(* Logix 5000 project; controller VET 1756-L62 rev 19.52; software revision 19.01; part 9 of 27 *)

        [46].Data.peso_f[8] := 50.0, [46].Data.peso_f[9] := 43.6, [46].Data.peso_f[10] := 35.0, [46].Data.peso_f[11] := 12.0, [46].Data.peso_f[12] := 60.0, [46].Data.peso_f[13] := 56.0, [46].Data.peso_f[14] := 25.0, [46].Data.peso_f[15] := 90.0, [46].Data.peso_r[0] := 332.00415, [46].Data.peso_r[1] := 319.90973, [46].Data.peso_r[2] := 285.3365, [46].Data.peso_r[3] := 180.5769, [46].Data.peso_r[4] := 159.76408, [46].Data.peso_r[5] := 109.9774, [46].Data.peso_r[6] := 90.60315, [46].Data.peso_r[7] := 90.27219, [46].Data.peso_r[8] := 50.001286, [46].Data.peso_r[9] := 43.602726, [46].Data.peso_r[10] := 34.989906, [46].Data.peso_r[11] := 11.96817, [46].Data.peso_r[12] := 59.986206, [46].Data.peso_r[13] := 56.00316, [46].Data.peso_r[14] := 25.010452, [46].Data.peso_r[15] := 89.91622, [46].Data.tolva[0] := 3, [46].Data.tolva[1] := 4, [46].Data.tolva[2] := 10, [46].Data.tolva[3] := 12, [46].Data.tolva[4] := 6, [46].Data.tolva[5] := 7, [46].Data.tolva[6] := 14, [46].Data.tolva[7] := 15, [46].Data.tolva[8] := 18, [46].Data.tolva[9] := 20, [46].Data.tolva[10] := 22, [46].Data.tolva[11] := 24, [46].Data.tolva[12] := 27, [46].Data.tolva[13] := 29, [46].Data.tolva[14] := 31, [46].Data.tolva[15] := 38, [46].Data.lugar[0] := 1, [46].Data.lugar[1] := 1, [46].Data.lugar[2] := 1, [46].Data.lugar[3] := 1, [46].Data.lugar[4] := 2, [46].Data.lugar[5] := 2, [46].Data.lugar[6] := 2, [46].Data.lugar[7] := 2, [46].Data.lugar[8] := 3, [46].Data.lugar[9] := 3, [46].Data.lugar[10] := 3, [46].Data.lugar[11] := 3, [46].Data.lugar[12] := 4, [46].Data.lugar[13] := 4, [46].Data.lugar[14] := 4, [46].Data.lugar[15] := 6, [46].Data.flags[0] := 5, [46].Data.flags[1] := 5, [46].Data.flags[2] := 5, [46].Data.flags[3] := 5,
        [46].Data.flags[4] := 5, [46].Data.flags[5] := 5, [46].Data.flags[6] := 5, [46].Data.flags[7] := 5, [46].Data.flags[8] := 5, [46].Data.flags[9] := 5, [46].Data.flags[10] := 5, [46].Data.flags[11] := 5, [46].Data.flags[12] := 5, [46].Data.flags[13] := 5, [46].Data.flags[14] := 5, [46].Data.flags[15] := 5, [46].Data.fecha_i[0] := 19980102, [46].Data.fecha_i[1] := 19980102, [46].Data.fecha_i[2] := 19980102, [46].Data.fecha_i[3] := 19980102, [46].Data.fecha_i[4] := 19980102, [46].Data.fecha_i[5] := 19980102, [46].Data.fecha_i[6] := 19980102, [46].Data.fecha_i[7] := 19980102, [46].Data.fecha_i[8] := 19980102, [46].Data.fecha_i[9] := 19980102, [46].Data.fecha_i[10] := 19980102, [46].Data.fecha_i[11] := 19980102, [46].Data.fecha_i[12] := 19980102, [46].Data.fecha_i[13] := 19980102, [46].Data.fecha_i[14] := 19980102, [46].Data.fecha_i[15] := 19980102, [46].Data.fecha_f[0] := 19980102, [46].Data.fecha_f[1] := 19980102, [46].Data.fecha_f[2] := 19980102, [46].Data.fecha_f[3] := 19980102, [46].Data.fecha_f[4] := 19980102, [46].Data.fecha_f[5] := 19980102, [46].Data.fecha_f[6] := 19980102, [46].Data.fecha_f[7] := 19980102, [46].Data.fecha_f[8] := 19980102, [46].Data.fecha_f[9] := 19980102, [46].Data.fecha_f[10] := 19980102, [46].Data.fecha_f[11] := 19980102, [46].Data.fecha_f[12] := 19980102, [46].Data.fecha_f[13] := 19980102, [46].Data.fecha_f[14] := 19980102, [46].Data.fecha_f[15] := 19980102, [46].Data.hora_i[0] := 22451016, [46].Data.hora_i[1] := 22452601, [46].Data.hora_i[2] := 22454141, [46].Data.hora_i[3] := 22455546, [46].Data.hora_i[4] := 22451016, [46].Data.hora_i[5] := 22452781, [46].Data.hora_i[6] := 22453811, [46].Data.hora_i[7] := 22455416, [46].Data.hora_i[8] := 22451016, [46].Data.hora_i[9] := 22465331, [46].Data.hora_i[10] := 22482366, [46].Data.hora_i[11] := 22493681, [46].Data.hora_i[12] := 22451016, [46].Data.hora_i[13] := 22471706, [46].Data.hora_i[14] := 22491621, [46].Data.hora_i[15] := 22503341,
        [46].Data.hora_f[0] := 22452581, [46].Data.hora_f[1] := 22454121, [46].Data.hora_f[2] := 22455526, [46].Data.hora_f[3] := 22460531, [46].Data.hora_f[4] := 22452761, [46].Data.hora_f[5] := 22453791, [46].Data.hora_f[6] := 22455396, [46].Data.hora_f[7] := 22460296, [46].Data.hora_f[8] := 22465311, [46].Data.hora_f[9] := 22482346, [46].Data.hora_f[10] := 22493661, [46].Data.hora_f[11] := 22500376, [46].Data.hora_f[12] := 22471686, [46].Data.hora_f[13] := 22491601, [46].Data.hora_f[14] := 22501286, [46].Data.hora_f[15] := 22512556, [47].Head.folio := 48, [47].Head.orden := -4, [47].Head.formula := 'DUMMY$00$00$00$00$00', [47].Head.correlativo := 8, [47].Head.total_batch := 10, [47].Head.peso_teorico := 1939.6, [47].Data.codigo[0] := 51, [47].Data.codigo[1] := 53, [47].Data.codigo[2] := 55, [47].Data.codigo[3] := 57, [47].Data.codigo[4] := 59, [47].Data.codigo[5] := 60, [47].Data.codigo[6] := 63, [47].Data.codigo[7] := 64, [47].Data.codigo[8] := 67, [47].Data.codigo[9] := 69, [47].Data.codigo[10] := 71, [47].Data.codigo[11] := 73, [47].Data.codigo[12] := 75, [47].Data.codigo[13] := 77, [47].Data.codigo[14] := 79, [47].Data.codigo[15] := 81, [47].Data.peso_f[0] := 333.0, [47].Data.peso_f[1] := 320.0, [47].Data.peso_f[2] := 285.0, [47].Data.peso_f[3] := 180.0, [47].Data.peso_f[4] := 160.0, [47].Data.peso_f[5] := 110.0, [47].Data.peso_f[6] := 90.0, [47].Data.peso_f[7] := 90.0, [47].Data.peso_f[8] := 50.0, [47].Data.peso_f[9] := 43.6, [47].Data.peso_f[10] := 35.0, [47].Data.peso_f[11] := 12.0, [47].Data.peso_f[12] := 60.0, [47].Data.peso_f[13] := 56.0, [47].Data.peso_f[14] := 25.0, [47].Data.peso_f[15] := 90.0, [47].Data.peso_r[0] := 334.1721, [47].Data.peso_r[1] := 319.58975, [47].Data.peso_r[2] := 284.6056, [47].Data.peso_r[3] := 180.28247, [47].Data.peso_r[4] := 159.7642, [47].Data.peso_r[5] := 109.9774,
        [47].Data.peso_r[6] := 90.59973, [47].Data.peso_r[7] := 91.76578, [47].Data.peso_r[8] := 50.000805, [47].Data.peso_r[9] := 43.602703, [47].Data.peso_r[10] := 34.989876, [47].Data.peso_r[11] := 12.01152, [47].Data.peso_r[12] := 60.010212, [47].Data.peso_r[13] := 56.003162, [47].Data.peso_r[14] := 25.01043, [47].Data.peso_r[15] := 90.216225, [47].Data.tolva[0] := 3, [47].Data.tolva[1] := 4, [47].Data.tolva[2] := 10, [47].Data.tolva[3] := 12, [47].Data.tolva[4] := 6, [47].Data.tolva[5] := 7, [47].Data.tolva[6] := 14, [47].Data.tolva[7] := 15, [47].Data.tolva[8] := 18, [47].Data.tolva[9] := 20, [47].Data.tolva[10] := 22, [47].Data.tolva[11] := 24, [47].Data.tolva[12] := 27, [47].Data.tolva[13] := 29, [47].Data.tolva[14] := 31, [47].Data.tolva[15] := 38, [47].Data.lugar[0] := 1, [47].Data.lugar[1] := 1, [47].Data.lugar[2] := 1, [47].Data.lugar[3] := 1, [47].Data.lugar[4] := 2, [47].Data.lugar[5] := 2, [47].Data.lugar[6] := 2, [47].Data.lugar[7] := 2, [47].Data.lugar[8] := 3, [47].Data.lugar[9] := 3, [47].Data.lugar[10] := 3, [47].Data.lugar[11] := 3, [47].Data.lugar[12] := 4, [47].Data.lugar[13] := 4, [47].Data.lugar[14] := 4, [47].Data.lugar[15] := 6, [47].Data.flags[0] := 5, [47].Data.flags[1] := 5, [47].Data.flags[2] := 5, [47].Data.flags[3] := 5, [47].Data.flags[4] := 5, [47].Data.flags[5] := 5, [47].Data.flags[6] := 5, [47].Data.flags[7] := 5, [47].Data.flags[8] := 5, [47].Data.flags[9] := 5, [47].Data.flags[10] := 5, [47].Data.flags[11] := 5, [47].Data.flags[12] := 5, [47].Data.flags[13] := 5, [47].Data.flags[14] := 5, [47].Data.flags[15] := 5, [47].Data.fecha_i[0] := 19980102, [47].Data.fecha_i[1] := 19980102,
        [47].Data.fecha_i[2] := 19980102, [47].Data.fecha_i[3] := 19980102, [47].Data.fecha_i[4] := 19980102, [47].Data.fecha_i[5] := 19980102, [47].Data.fecha_i[6] := 19980102, [47].Data.fecha_i[7] := 19980102, [47].Data.fecha_i[8] := 19980102, [47].Data.fecha_i[9] := 19980102, [47].Data.fecha_i[10] := 19980102, [47].Data.fecha_i[11] := 19980102, [47].Data.fecha_i[12] := 19980102, [47].Data.fecha_i[13] := 19980102, [47].Data.fecha_i[14] := 19980102, [47].Data.fecha_i[15] := 19980102, [47].Data.fecha_f[0] := 19980102, [47].Data.fecha_f[1] := 19980102, [47].Data.fecha_f[2] := 19980102, [47].Data.fecha_f[3] := 19980102, [47].Data.fecha_f[4] := 19980102, [47].Data.fecha_f[5] := 19980102, [47].Data.fecha_f[6] := 19980102, [47].Data.fecha_f[7] := 19980102, [47].Data.fecha_f[8] := 19980102, [47].Data.fecha_f[9] := 19980102, [47].Data.fecha_f[10] := 19980102, [47].Data.fecha_f[11] := 19980102, [47].Data.fecha_f[12] := 19980102, [47].Data.fecha_f[13] := 19980102, [47].Data.fecha_f[14] := 19980102, [47].Data.fecha_f[15] := 19980102, [47].Data.hora_i[0] := 22522096, [47].Data.hora_i[1] := 22523686, [47].Data.hora_i[2] := 22525226, [47].Data.hora_i[3] := 22530631, [47].Data.hora_i[4] := 22522096, [47].Data.hora_i[5] := 22523861, [47].Data.hora_i[6] := 22524891, [47].Data.hora_i[7] := 22541271, [47].Data.hora_i[8] := 22522096, [47].Data.hora_i[9] := 22540411, [47].Data.hora_i[10] := 22553446, [47].Data.hora_i[11] := 22564761, [47].Data.hora_i[12] := 22522096, [47].Data.hora_i[13] := 22542786, [47].Data.hora_i[14] := 22562701, [47].Data.hora_i[15] := 22574421, [47].Data.hora_f[0] := 22523666, [47].Data.hora_f[1] := 22525206, [47].Data.hora_f[2] := 22530611, [47].Data.hora_f[3] := 22531616, [47].Data.hora_f[4] := 22523841, [47].Data.hora_f[5] := 22524871, [47].Data.hora_f[6] := 22541251, [47].Data.hora_f[7] := 22543396, [47].Data.hora_f[8] := 22540391, [47].Data.hora_f[9] := 22553426, [47].Data.hora_f[10] := 22564741, [47].Data.hora_f[11] := 22571461, [47].Data.hora_f[12] := 22542766, [47].Data.hora_f[13] := 22562681,
        [47].Data.hora_f[14] := 22572366, [47].Data.hora_f[15] := 22583656, [48].Head.folio := 49, [48].Head.orden := -4, [48].Head.formula := 'DUMMY$00$00$00$00$00', [48].Head.correlativo := 9, [48].Head.total_batch := 10, [48].Head.peso_teorico := 1939.6, [48].Data.codigo[0] := 51, [48].Data.codigo[1] := 53, [48].Data.codigo[2] := 55, [48].Data.codigo[3] := 57, [48].Data.codigo[4] := 59, [48].Data.codigo[5] := 60, [48].Data.codigo[6] := 63, [48].Data.codigo[7] := 64, [48].Data.codigo[8] := 67, [48].Data.codigo[9] := 69, [48].Data.codigo[10] := 71, [48].Data.codigo[11] := 73, [48].Data.codigo[12] := 75, [48].Data.codigo[13] := 77, [48].Data.codigo[14] := 79, [48].Data.codigo[15] := 81, [48].Data.peso_f[0] := 333.0, [48].Data.peso_f[1] := 320.0, [48].Data.peso_f[2] := 285.0, [48].Data.peso_f[3] := 180.0, [48].Data.peso_f[4] := 160.0, [48].Data.peso_f[5] := 110.0, [48].Data.peso_f[6] := 90.0, [48].Data.peso_f[7] := 90.0, [48].Data.peso_f[8] := 50.0, [48].Data.peso_f[9] := 43.6, [48].Data.peso_f[10] := 35.0, [48].Data.peso_f[11] := 12.0, [48].Data.peso_f[12] := 60.0, [48].Data.peso_f[13] := 56.0, [48].Data.peso_f[14] := 25.0, [48].Data.peso_f[15] := 90.0, [48].Data.peso_r[0] := 333.78995, [48].Data.peso_r[1] := 320.86465, [48].Data.peso_r[2] := 284.5542, [48].Data.peso_r[3] := 180.89838, [48].Data.peso_r[4] := 161.07552, [48].Data.peso_r[5] := 109.51335, [48].Data.peso_r[6] := 89.659424, [48].Data.peso_r[7] := 89.651245, [48].Data.peso_r[8] := 50.02211, [48].Data.peso_r[9] := 43.61187, [48].Data.peso_r[10] := 35.014, [48].Data.peso_r[11] := 12.01828, [48].Data.peso_r[12] := 60.01018, [48].Data.peso_r[13] := 56.003117, [48].Data.peso_r[14] := 25.012413, [48].Data.peso_r[15] := 89.91622, [48].Data.tolva[0] := 3, [48].Data.tolva[1] := 4, [48].Data.tolva[2] := 10, [48].Data.tolva[3] := 12,
        [48].Data.tolva[4] := 6, [48].Data.tolva[5] := 7, [48].Data.tolva[6] := 14, [48].Data.tolva[7] := 15, [48].Data.tolva[8] := 18, [48].Data.tolva[9] := 20, [48].Data.tolva[10] := 22, [48].Data.tolva[11] := 24, [48].Data.tolva[12] := 27, [48].Data.tolva[13] := 29, [48].Data.tolva[14] := 31, [48].Data.tolva[15] := 38, [48].Data.lugar[0] := 1, [48].Data.lugar[1] := 1, [48].Data.lugar[2] := 1, [48].Data.lugar[3] := 1, [48].Data.lugar[4] := 2, [48].Data.lugar[5] := 2, [48].Data.lugar[6] := 2, [48].Data.lugar[7] := 2, [48].Data.lugar[8] := 3, [48].Data.lugar[9] := 3, [48].Data.lugar[10] := 3, [48].Data.lugar[11] := 3, [48].Data.lugar[12] := 4, [48].Data.lugar[13] := 4, [48].Data.lugar[14] := 4, [48].Data.lugar[15] := 6, [48].Data.flags[0] := 5, [48].Data.flags[1] := 5, [48].Data.flags[2] := 5, [48].Data.flags[3] := 5, [48].Data.flags[4] := 5, [48].Data.flags[5] := 5, [48].Data.flags[6] := 5, [48].Data.flags[7] := 5, [48].Data.flags[8] := 5, [48].Data.flags[9] := 5, [48].Data.flags[10] := 5, [48].Data.flags[11] := 5, [48].Data.flags[12] := 5, [48].Data.flags[13] := 5, [48].Data.flags[14] := 5, [48].Data.flags[15] := 5, [48].Data.fecha_i[0] := 19980102, [48].Data.fecha_i[1] := 19980102, [48].Data.fecha_i[2] := 19980102, [48].Data.fecha_i[3] := 19980102, [48].Data.fecha_i[4] := 19980102, [48].Data.fecha_i[5] := 19980102, [48].Data.fecha_i[6] := 19980102, [48].Data.fecha_i[7] := 19980102, [48].Data.fecha_i[8] := 19980102, [48].Data.fecha_i[9] := 19980102, [48].Data.fecha_i[10] := 19980102, [48].Data.fecha_i[11] := 19980102, [48].Data.fecha_i[12] := 19980102, [48].Data.fecha_i[13] := 19980102, [48].Data.fecha_i[14] := 19980102, [48].Data.fecha_i[15] := 19980102,
        [48].Data.fecha_f[0] := 19980102, [48].Data.fecha_f[1] := 19980102, [48].Data.fecha_f[2] := 19980102, [48].Data.fecha_f[3] := 19980102, [48].Data.fecha_f[4] := 19980102, [48].Data.fecha_f[5] := 19980102, [48].Data.fecha_f[6] := 19980102, [48].Data.fecha_f[7] := 19980102, [48].Data.fecha_f[8] := 19980102, [48].Data.fecha_f[9] := 19980102, [48].Data.fecha_f[10] := 19980102, [48].Data.fecha_f[11] := 19980102, [48].Data.fecha_f[12] := 19980102, [48].Data.fecha_f[13] := 19980102, [48].Data.fecha_f[14] := 19980102, [48].Data.fecha_f[15] := 19980102, [48].Data.hora_i[0] := 22574426, [48].Data.hora_i[1] := 22580016, [48].Data.hora_i[2] := 22581556, [48].Data.hora_i[3] := 22582961, [48].Data.hora_i[4] := 22574426, [48].Data.hora_i[5] := 22580691, [48].Data.hora_i[6] := 22581716, [48].Data.hora_i[7] := 22582616, [48].Data.hora_i[8] := 22574426, [48].Data.hora_i[9] := 22592741, [48].Data.hora_i[10] := 23005776, [48].Data.hora_i[11] := 23021091, [48].Data.hora_i[12] := 22574426, [48].Data.hora_i[13] := 22595111, [48].Data.hora_i[14] := 23015026, [48].Data.hora_i[15] := 23030746, [48].Data.hora_f[0] := 22575996, [48].Data.hora_f[1] := 22581536, [48].Data.hora_f[2] := 22582941, [48].Data.hora_f[3] := 22583951, [48].Data.hora_f[4] := 22580671, [48].Data.hora_f[5] := 22581696, [48].Data.hora_f[6] := 22582596, [48].Data.hora_f[7] := 22583496, [48].Data.hora_f[8] := 22592721, [48].Data.hora_f[9] := 23005756, [48].Data.hora_f[10] := 23021071, [48].Data.hora_f[11] := 23023791, [48].Data.hora_f[12] := 22595091, [48].Data.hora_f[13] := 23015006, [48].Data.hora_f[14] := 23024691, [48].Data.hora_f[15] := 23035961, [49].Head.folio := 50, [49].Head.orden := -4, [49].Head.formula := 'DUMMY$00$00$00$00$00', [49].Head.correlativo := 10, [49].Head.total_batch := 10, [49].Head.peso_teorico := 1939.6, [49].Data.codigo[0] := 51, [49].Data.codigo[1] := 53, [49].Data.codigo[2] := 55, [49].Data.codigo[3] := 57, [49].Data.codigo[4] := 59, [49].Data.codigo[5] := 60,
        [49].Data.codigo[6] := 63, [49].Data.codigo[7] := 64, [49].Data.codigo[8] := 67, [49].Data.codigo[9] := 69, [49].Data.codigo[10] := 71, [49].Data.codigo[11] := 73, [49].Data.codigo[12] := 75, [49].Data.codigo[13] := 77, [49].Data.codigo[14] := 79, [49].Data.codigo[15] := 81, [49].Data.peso_f[0] := 333.0, [49].Data.peso_f[1] := 320.0, [49].Data.peso_f[2] := 285.0, [49].Data.peso_f[3] := 180.0, [49].Data.peso_f[4] := 160.0, [49].Data.peso_f[5] := 110.0, [49].Data.peso_f[6] := 90.0, [49].Data.peso_f[7] := 90.0, [49].Data.peso_f[8] := 50.0, [49].Data.peso_f[9] := 43.6, [49].Data.peso_f[10] := 35.0, [49].Data.peso_f[11] := 12.0, [49].Data.peso_f[12] := 60.0, [49].Data.peso_f[13] := 56.0, [49].Data.peso_f[14] := 25.0, [49].Data.peso_f[15] := 90.0, [49].Data.peso_r[0] := 332.00412, [49].Data.peso_r[1] := 319.9097, [49].Data.peso_r[2] := 285.33063, [49].Data.peso_r[3] := 180.57697, [49].Data.peso_r[4] := 159.76414, [49].Data.peso_r[5] := 110.49193, [49].Data.peso_r[6] := 90.60315, [49].Data.peso_r[7] := 90.78711, [49].Data.peso_r[8] := 50.00127, [49].Data.peso_r[9] := 43.58846, [49].Data.peso_r[10] := 35.014, [49].Data.peso_r[11] := 12.01828, [49].Data.peso_r[12] := 59.986187, [49].Data.peso_r[13] := 56.003162, [49].Data.peso_r[14] := 25.010452, [49].Data.peso_r[15] := 89.916214, [49].Data.tolva[0] := 3, [49].Data.tolva[1] := 4, [49].Data.tolva[2] := 10, [49].Data.tolva[3] := 12, [49].Data.tolva[4] := 6, [49].Data.tolva[5] := 7, [49].Data.tolva[6] := 14, [49].Data.tolva[7] := 15, [49].Data.tolva[8] := 18, [49].Data.tolva[9] := 20, [49].Data.tolva[10] := 22, [49].Data.tolva[11] := 24, [49].Data.tolva[12] := 27, [49].Data.tolva[13] := 29, [49].Data.tolva[14] := 31, [49].Data.tolva[15] := 38, [49].Data.lugar[0] := 1, [49].Data.lugar[1] := 1,
        [49].Data.lugar[2] := 1, [49].Data.lugar[3] := 1, [49].Data.lugar[4] := 2, [49].Data.lugar[5] := 2, [49].Data.lugar[6] := 2, [49].Data.lugar[7] := 2, [49].Data.lugar[8] := 3, [49].Data.lugar[9] := 3, [49].Data.lugar[10] := 3, [49].Data.lugar[11] := 3, [49].Data.lugar[12] := 4, [49].Data.lugar[13] := 4, [49].Data.lugar[14] := 4, [49].Data.lugar[15] := 6, [49].Data.flags[0] := 5, [49].Data.flags[1] := 5, [49].Data.flags[2] := 5, [49].Data.flags[3] := 5, [49].Data.flags[4] := 5, [49].Data.flags[5] := 5, [49].Data.flags[6] := 5, [49].Data.flags[7] := 5, [49].Data.flags[8] := 5, [49].Data.flags[9] := 5, [49].Data.flags[10] := 5, [49].Data.flags[11] := 5, [49].Data.flags[12] := 5, [49].Data.flags[13] := 5, [49].Data.flags[14] := 5, [49].Data.flags[15] := 5, [49].Data.fecha_i[0] := 20140515, [49].Data.fecha_i[1] := 20140515, [49].Data.fecha_i[2] := 20140515, [49].Data.fecha_i[3] := 20140515, [49].Data.fecha_i[4] := 20140515, [49].Data.fecha_i[5] := 20140515, [49].Data.fecha_i[6] := 20140515, [49].Data.fecha_i[7] := 20140515, [49].Data.fecha_i[8] := 20140515, [49].Data.fecha_i[9] := 20140515, [49].Data.fecha_i[10] := 20140515, [49].Data.fecha_i[11] := 20140515, [49].Data.fecha_i[12] := 20140515, [49].Data.fecha_i[13] := 20140515, [49].Data.fecha_i[14] := 20140515, [49].Data.fecha_i[15] := 20140515, [49].Data.fecha_f[0] := 20140515, [49].Data.fecha_f[1] := 20140515, [49].Data.fecha_f[2] := 20140515, [49].Data.fecha_f[3] := 20140515, [49].Data.fecha_f[4] := 20140515, [49].Data.fecha_f[5] := 20140515, [49].Data.fecha_f[6] := 20140515, [49].Data.fecha_f[7] := 20140515, [49].Data.fecha_f[8] := 20140515, [49].Data.fecha_f[9] := 20140515, [49].Data.fecha_f[10] := 20140515, [49].Data.fecha_f[11] := 20140515, [49].Data.fecha_f[12] := 20140515, [49].Data.fecha_f[13] := 20140515,
        [49].Data.fecha_f[14] := 20140515, [49].Data.fecha_f[15] := 20140515, [49].Data.hora_i[0] := 13231208, [49].Data.hora_i[1] := 13232798, [49].Data.hora_i[2] := 13234338, [49].Data.hora_i[3] := 13235743, [49].Data.hora_i[4] := 13231208, [49].Data.hora_i[5] := 13232978, [49].Data.hora_i[6] := 13234008, [49].Data.hora_i[7] := 13264413, [49].Data.hora_i[8] := 13231208, [49].Data.hora_i[9] := 13245523, [49].Data.hora_i[10] := 13262553, [49].Data.hora_i[11] := 13273868, [49].Data.hora_i[12] := 13231208, [49].Data.hora_i[13] := 13251898, [49].Data.hora_i[14] := 13271788, [49].Data.hora_i[15] := 13305218, [49].Data.hora_f[0] := 13232778, [49].Data.hora_f[1] := 13234318, [49].Data.hora_f[2] := 13235723, [49].Data.hora_f[3] := 13240728, [49].Data.hora_f[4] := 13232958, [49].Data.hora_f[5] := 13233988, [49].Data.hora_f[6] := 13264393, [49].Data.hora_f[7] := 13303843, [49].Data.hora_f[8] := 13245503, [49].Data.hora_f[9] := 13262533, [49].Data.hora_f[10] := 13273848, [49].Data.hora_f[11] := 13280568, [49].Data.hora_f[12] := 13251878, [49].Data.hora_f[13] := 13271768, [49].Data.hora_f[14] := 13281488, [49].Data.hora_f[15] := 13314433);
   borrar : DINT[100] := ([0] := 262822, [1] := 17, [2] := 1477, [3] := 8423, [4] := 4406, [5] := 161022, [6] := 458752, [7] := 589841, [10] := 2, [11] := 3, [13] := 612380685, [14] := 37, [15] := 9194, [16] := 11, [17] := 48, [18] := 1009, [19] := 34, [22] := 1, [23] := 452, [24] := 4096, [26] := 13, [27] := 64, [30] := 16, [31] := 21000, [32] := 288, [33] := 7, [34] := 131313, [35] := 19, [36] := 3, [37] := 672, [38] := 237, [41] := 701600, [43] := 16, [47] := 59, [48] := 65518, [50] := 128, [51] := 72, [54] := 1, [55] := 1, [56] := 15, [58] := 4, [60] := 6291460, [61] := 28, [64] := 32767, [65] := 65535, [67] := 1, [68] := 11, [73] := 32768, [75] := 38, [80] := 2097152, [91] := 1, [92] := 1256256, [97] := 5, [99] := 870);
        [37].20   // Copy BatchDMM[6] -> BatchBUFF[3]
        [0].0   // Main
        [0].2   // Enable V0
        [0].18   // Bypass IO
        [1].1   // Simulación
        [6].1   // Cerrar
        [6].2   // Abrir
        [6].3   // Cerrar
        [6].4   // Abrir
        [37].21   // Copy Batch[2] -> Batch[0]
        [6].5   // Cerrar
        [6].6   // Abrir
        [6].7   // Cerrar
        [8].0   // Forma S88
        [11].3   // _
        [0].1   // Simulacion IO
        [0].19   // Exec Startup
        [80].21   // IO MOLIENDA
        [0]   // _
        [1]   // _
        [3]   // _
        [4]   // _
        [6]   // _
        [7]   // _
        [67].0   // Nuevos Complete
   comandos : DINT[10] := ([0] := 1, [1] := 127);
        [0].0   // Recibir Batch
        [1]   // Comandos Generales
        [0].3   // Retornar Batch
        [0]   // Comandos Batch
        [0].1   // Envío Automático de Batch
        [0].2   // Envío Manual de Batch
        [0].4   // Recibiendo Batch (DB)
   corriente : REAL[40] := ([0] := 15.0, [1] := 9.0);
        [0]   // Corriente Mezcladora
        [1]   // Corriente Elevador Despacho
        [2]   // Corriente Elevador Abastecimiento
   db_input_cola : cola_almacenes;
   db_input_cola_batch_res : DINT;
   db_input_cola_flag : BOOL;
   dosificador : dosif_struct[20] := ([0].estado_phases._idle := 1, [1].estado_phases._idle := 1, [2].estado_phases._idle := 1, [3].estado_phases._idle := 1, [4].estado_phases._idle := 1, [5].peso_terreno := 89.916214, [5].estado_phases._idle := 1);
        [5]   // Líquidos 1
        [1]   // Midis 1
        [4]   // Manuales
        [2]   // Micros 1
        [3]   // Micros 2
        [0]   // Macros 1
   Dosificar_LIQ_01 : PHASE := (State := 64, Idle := 1);
   Dosificar_MAC_01 : PHASE := (State := 64, Idle := 1);
   Dosificar_MAN_01 : PHASE := (State := 64, Idle := 1);
   Dosificar_MIC_01 : PHASE := (State := 64, Idle := 1);
   Dosificar_MIC_02 : PHASE := (State := 64, Idle := 1);
   Dosificar_MID_01 : PHASE := (State := 64, Idle := 1);
   DRT : DRTs[10] := ([0].InputPos := 4, [0].CmdPos := 3, [0].ConfPos := 3, [0].RealPos := 3, [0].TotalPos := 6, [1].InputPos := 64, [1].CmdPos := 7, [1].ConfPos := 7, [1].RealPos := 7, [1].TotalPos := 8, [2].InputPos := 4, [2].CmdPos := 3, [2].ConfPos := 3, [2].RealPos := 3, [2].TotalPos := 8, [3].InputPos := 2, [3].CmdPos := 2, [3].ConfPos := 2, [3].RealPos := 2, [3].TotalPos := 4);
   fecha_plc : DINT := 20140515;
   flujometro : flujometro[5] := ([0].scale_total.Input := 89.916214, [0].scale_total.InHigh := 1.0, [0].scale_total.OutHigh := 1.0, [0].scale_total.Output := 89.916214, [0].total := 10616.379, [0].total_batch := 89.916214, [0].total_scaled := 10616.379, [0].total_scaled_batch := 89.916214, [0].T.PRE := 10000000, [0].set_in := 1.0, [0].set_out := 1.0, [0].input := 4000, [0].delta_t := 48, [1].scale_flujo.Input := 4000.0, [1].scale_flujo.InLow := 4000.0, [1].scale_flujo.InHigh := 20000.0, [1].scale_flujo.OutHigh := 4.0, [1].flujo := -1.0);
        [0].AUX.2   // Borrar Acumulado Batch
   hora_plc : DINT := 18464533;
   peso_tolva : REAL[80] := ([37] := 6814.857, [38] := 89.916214);
        [33]   // Peso Macros
        [34]   // Peso Midis
        [35]   // Peso Micros 1
        [36]   // Peso Micros 2
        [0]   // dummy
        [37]   // Peso Liq 1
   Set_Global : DINT[20] := ([0] := 300, [1] := 2, [2] := 2, [3] := 1, [6] := 1, [8] := 5);
        [6]   // N° de Líneas
        [0]   // Nº de Equipos
        [1]   // Nº de Selectores
        [2]   // Nº de Origenes
        [3]   // N° de Línea 1
        [4]   // N° de Línea 2
        [5]   // N° de Línea 3
   SetDInt : DINT[500] := ([0] := 5, [1] := 300, [2] := 100, [3] := 96, [4] := 3, [5] := 200, [6] := 27, [7] := 100, [8] := 18, [9] := 45, [10] := 80, [11] := 40, [12] := 18, [13] := 20, [14] := 31, [15] := 32, [16] := 120, [17] := 19, [18] := 10, [20] := 4, [21] := 150, [22] := 180, [23] := 150, [24] := 180, [25] := 120, [26] := 120, [27] := 20, [28] := 7, [29] := 10, [30] := 10, [31] := 6, [32] := 1, [33] := 2, [34] := 3, [35] := 4, [36] := 40, [37] := 40, [38] := 500, [40] := 30000, [41] := 1, [42] := 10, [43] := 546, [44] := 2, [46] := 14, [47] := 26, [48] := 32, [50] := 160);
        [11]   // Número Máximo de Ingredientes
        [10]   // Número Máximo de Tolvas
   simulacion : BOOL := 1;
   SS_Comun : Soft_Starter := (Idx_Equipo[0] := 326, Idx_Equipo[1] := 325, Partiendo := 1, Flags := 1, Tpo_Espera.PRE := 15000, Tpos_Grl[0].PRE := 3000);
   SSvar : set_variables := (setD[0] := 13, i0 := 9, i2 := 283, i3 := 1, i5 := 10, i6 := 7);
   Tab_ODS : Tab_O_D_Orig := (O[1].D[1].S[1] := 1, O[1].D[2].S[1] := 2, O[1].D[3].S[1] := 3, O[1].D[4].S[1] := 4, O[1].D[5].S[1] := 5, O[1].D[6].S[1] := 6, O[1].D[7].S[1] := 7, O[1].D[8].S[1] := 8, O[1].D[9].S[1] := 9, O[1].D[10].S[1] := 10, O[1].D[11].S[1] := 11, O[1].D[12].S[1] := 12, O[1].D[13].S[1] := 13, O[1].D[14].S[1] := 14, O[1].D[15].S[1] := 15, O[1].D[16].S[1] := 16, O[1].Eqp[1] := 20, O[1].Eqp[2] := 21, O[1].Eqp[3] := 22, O[1].Eqp[4] := 23, O[1].Eqp[5] := 24, O[1].Eqp[6] := 25, O[1].Eqp[7] := 26, O[1].Eqp[8] := 27, O[1].Eqp[9] := 28, O[1].Eqp[10] := 29, O[1].Eqp[11] := 30, O[1].Eqp[12] := 31, O[1].Eqp[13] := 32, O[1].Eqp[14] := 33, O[1].Eqp[15] := 34, O[1].Eqp[16] := 35, O[2].D[1].S[2] := 1, O[2].D[2].S[2] := 2, O[2].Eqp[1] := 140, O[2].Eqp[2] := 150);   // Tabla Origen Destino
   TabBin : Bins_Setup := (c.id[1] := 1, c.id[2] := 2, c.id[3] := 3, c.id[4] := 4, c.id[5] := 5, c.id[6] := 6, c.id[7] := 7, c.id[8] := 8, c.id[9] := 9, c.id[10] := 10, c.id[11] := 11, c.id[12] := 12, c.id[13] := 13, c.id[14] := 14, c.id[15] := 15, c.id[16] := 16, c.id[17] := 17, c.id[18] := 18, c.id[19] := 19, c.id[20] := 20, c.id[21] := 21, c.id[22] := 22, c.id[23] := 23, c.id[24] := 24, c.id[25] := 25, c.id[26] := 26, c.id[27] := 27, c.id[28] := 28, c.id[29] := 29, c.id[30] := 30, c.id[31] := 31, c.id[32] := 32, c.id[33] := 33, c.id[34] := 34, c.id[35] := 35, c.id[36] := 36, c.id[37] := 37, c.id[38] := 38, c.id[39] := 39, c.id[40] := 40, c.id[41] := 41, c.tolva[1] := 1, c.tolva[2] := 1, c.tolva[3] := 2, c.tolva[4] := 3, c.tolva[5] := 4, c.tolva[6] := 5, c.tolva[7] := 6, c.tolva[8] := 7, c.tolva[9] := 8, c.tolva[10] := 9, c.tolva[11] := 10, c.tolva[12] := 11, c.tolva[13] := 12, c.tolva[14] := 13, c.tolva[15] := 14, c.tolva[16] := 15, c.tolva[17] := 16, c.tolva[18] := 17, c.tolva[19] := 18,
        c.tolva[20] := 19, c.tolva[21] := 20, c.tolva[22] := 21, c.tolva[23] := 22, c.tolva[24] := 23, c.tolva[25] := 33, c.tolva[26] := 24, c.tolva[27] := 25, c.tolva[28] := 26, c.tolva[29] := 27, c.tolva[30] := 28, c.tolva[31] := 29, c.tolva[32] := 30, c.tolva[33] := 1, c.tolva[34] := 1, c.tolva[35] := 1, c.tolva[36] := 1, c.tolva[37] := 1, c.tolva[38] := 1, c.tolva[39] := 31, c.tolva[40] := 32, c.tolva[41] := 33, c.n_tolva[1] := 2, c.n_tolva[2] := 20, c.n_tolva[3] := 21, c.n_tolva[4] := 22, c.n_tolva[5] := 23, c.n_tolva[6] := 24, c.n_tolva[7] := 25, c.n_tolva[8] := 26, c.n_tolva[9] := 27, c.n_tolva[10] := 28, c.n_tolva[11] := 29, c.n_tolva[12] := 30, c.n_tolva[13] := 31, c.n_tolva[14] := 32, c.n_tolva[15] := 34, c.n_tolva[16] := 35, c.n_tolva[17] := 36, c.n_tolva[18] := 60, c.n_tolva[19] := 61, c.n_tolva[20] := 62, c.n_tolva[21] := 63, c.n_tolva[22] := 64, c.n_tolva[23] := 65, c.n_tolva[24] := 66, c.n_tolva[25] := 74, c.n_tolva[26] := 67, c.n_tolva[27] := 68, c.n_tolva[28] := 69, c.n_tolva[29] := 70, c.n_tolva[30] := 71, c.n_tolva[31] := 72, c.n_tolva[32] := 73, c.n_tolva[33] := 110, c.n_tolva[34] := 112, c.n_tolva[35] := 114, c.n_tolva[36] := 116, c.n_tolva[37] := 129, c.n_tolva[38] := 120,
        c.n_tolva[39] := 132, c.n_tolva[40] := 140, c.n_tolva[41] := 150, c.equipo1[2] := 40, c.equipo1[3] := 41, c.equipo1[4] := 42, c.equipo1[5] := 43, c.equipo1[6] := 44, c.equipo1[7] := 45, c.equipo1[8] := 46, c.equipo1[9] := 47, c.equipo1[10] := 48, c.equipo1[11] := 49, c.equipo1[12] := 50, c.equipo1[13] := 51, c.equipo1[14] := 52, c.equipo1[15] := 53, c.equipo1[16] := 54, c.equipo1[17] := 55, c.equipo1[18] := 80, c.equipo1[19] := 81, c.equipo1[20] := 82, c.equipo1[21] := 83, c.equipo1[22] := 84, c.equipo1[23] := 85, c.equipo1[24] := 86, c.equipo1[25] := 94, c.equipo1[26] := 87, c.equipo1[27] := 88, c.equipo1[28] := 89, c.equipo1[29] := 90, c.equipo1[30] := 91, c.equipo1[31] := 92, c.equipo1[32] := 93, c.equipo1[38] := 123, c.equipo2[5] := 10, c.equipo2[6] := 11, c.equipo2[8] := 12, c.equipo2[11] := 13, c.equipo2[13] := 14, c.equipo2[17] := 15, c.equipo2[19] := 100, c.equipo2[21] := 101, c.equipo2[23] := 102, c.equipo2[27] := 103, c.equipo2[29] := 104, c.equipo2[31] := 105, c.equipo2[38] := 121, c.dosificador[2] := 1, c.dosificador[3] := 1, c.dosificador[4] := 1, c.dosificador[5] := 1, c.dosificador[6] := 2, c.dosificador[7] := 2, c.dosificador[8] := 2, c.dosificador[9] := 2, c.dosificador[10] := 1, c.dosificador[11] := 1, c.dosificador[12] := 1, c.dosificador[13] := 1,
        c.dosificador[14] := 2, c.dosificador[15] := 2, c.dosificador[16] := 2, c.dosificador[17] := 2, c.dosificador[18] := 3, c.dosificador[19] := 3, c.dosificador[20] := 3, c.dosificador[21] := 3, c.dosificador[22] := 3, c.dosificador[23] := 3, c.dosificador[24] := 3, c.dosificador[25] := 5, c.dosificador[26] := 4, c.dosificador[27] := 4, c.dosificador[28] := 4, c.dosificador[29] := 4, c.dosificador[30] := 4, c.dosificador[31] := 4, c.dosificador[32] := 4, c.dosificador[38] := 6, c.codigo[1] := 1, c.codigo[2] := 54, c.codigo[3] := 54, c.codigo[4] := 53, c.codigo[5] := 54, c.codigo[6] := 59, c.codigo[7] := 60, c.codigo[8] := 61, c.codigo[9] := 62, c.codigo[10] := 55, c.codigo[11] := 56, c.codigo[12] := 57, c.codigo[13] := 58, c.codigo[14] := 63, c.codigo[15] := 64, c.codigo[16] := 65, c.codigo[17] := 66, c.codigo[18] := 67, c.codigo[19] := 68, c.codigo[20] := 69, c.codigo[21] := 70, c.codigo[22] := 71, c.codigo[23] := 72, c.codigo[24] := 73, c.codigo[26] := 74, c.codigo[27] := 75, c.codigo[28] := 76, c.codigo[29] := 77, c.codigo[30] := 78, c.codigo[31] := 79, c.codigo[32] := 80, c.codigo[38] := 81, c.sql_codigo[1] := 1, c.sql_codigo[2] := 54, c.sql_codigo[3] := 54, c.sql_codigo[4] := 53, c.sql_codigo[5] := 54, c.sql_codigo[6] := 59, c.sql_codigo[7] := 60, c.sql_codigo[8] := 61,
        c.sql_codigo[9] := 62, c.sql_codigo[10] := 55, c.sql_codigo[11] := 56, c.sql_codigo[12] := 57, c.sql_codigo[13] := 58, c.sql_codigo[14] := 63, c.sql_codigo[15] := 64, c.sql_codigo[16] := 65, c.sql_codigo[17] := 66, c.sql_codigo[18] := 67, c.sql_codigo[19] := 68, c.sql_codigo[20] := 69, c.sql_codigo[21] := 70, c.sql_codigo[22] := 71, c.sql_codigo[23] := 72, c.sql_codigo[24] := 73, c.sql_codigo[26] := 74, c.sql_codigo[27] := 75, c.sql_codigo[28] := 76, c.sql_codigo[29] := 77, c.sql_codigo[30] := 78, c.sql_codigo[31] := 79, c.sql_codigo[32] := 80, c.sql_codigo[38] := 81, c.prioridad[2] := 2, c.prioridad[3] := 1, c.prioridad[4] := 1, c.prioridad[5] := 1, c.prioridad[6] := 1, c.prioridad[7] := 1, c.prioridad[8] := 1, c.prioridad[9] := 1, c.prioridad[10] := 1, c.prioridad[11] := 1, c.prioridad[12] := 1, c.prioridad[13] := 1, c.prioridad[14] := 1, c.prioridad[15] := 1, c.prioridad[16] := 1, c.prioridad[17] := 1, c.prioridad[18] := 1, c.prioridad[19] := 1, c.prioridad[20] := 1, c.prioridad[21] := 1, c.prioridad[22] := 1, c.prioridad[23] := 1, c.prioridad[24] := 1, c.prioridad[26] := 1, c.prioridad[27] := 1, c.prioridad[28] := 1, c.prioridad[29] := 1, c.prioridad[30] := 1, c.prioridad[31] := 1, c.prioridad[32] := 1, c.prioridad[38] := 1, d[0].t_espera[2] := 3000, d[0].t_espera[3] := 3000, d[0].t_espera[4] := 3000, d[0].t_espera[5] := 3000, d[0].t_espera[6] := 3000,
        d[0].t_espera[7] := 3000, d[0].t_espera[8] := 3000, d[0].t_espera[9] := 3000, d[0].t_espera[10] := 3000, d[0].t_espera[11] := 3000, d[0].t_espera[12] := 3000, d[0].t_espera[13] := 3000, d[0].t_espera[14] := 3000, d[0].t_espera[15] := 3000, d[0].t_espera[16] := 3000, d[0].t_espera[17] := 3000, d[0].t_espera[18] := 3000, d[0].t_espera[19] := 3000, d[0].t_espera[20] := 3000, d[0].t_espera[21] := 3000, d[0].t_espera[22] := 3000, d[0].t_espera[23] := 3000, d[0].t_espera[24] := 3000, d[0].t_espera[26] := 3000, d[0].t_espera[27] := 3000, d[0].t_espera[28] := 3000, d[0].t_espera[29] := 3000, d[0].t_espera[30] := 3000, d[0].t_espera[31] := 3000, d[0].t_espera[32] := 3000, d[0].t_espera[38] := 3000, d[0].t_pulso[2] := 10000, d[0].t_pulso[3] := 10000, d[0].t_pulso[4] := 10000, d[0].t_pulso[5] := 10000, d[0].t_pulso[6] := 10000, d[0].t_pulso[7] := 10000, d[0].t_pulso[8] := 10000, d[0].t_pulso[9] := 10000, d[0].t_pulso[10] := 10000, d[0].t_pulso[11] := 10000, d[0].t_pulso[12] := 10000, d[0].t_pulso[13] := 10000, d[0].t_pulso[14] := 10000, d[0].t_pulso[15] := 10000, d[0].t_pulso[16] := 10000, d[0].t_pulso[17] := 10000, d[0].t_pulso[18] := 6000, d[0].t_pulso[19] := 6000, d[0].t_pulso[20] := 6000, d[0].t_pulso[21] := 6000, d[0].t_pulso[22] := 6000, d[0].t_pulso[23] := 6000, d[0].t_pulso[24] := 6000, d[0].t_pulso[26] := 6000, d[0].t_pulso[27] := 6000, d[0].t_pulso[28] := 6000, d[0].t_pulso[29] := 6000, d[0].t_pulso[30] := 6000, d[0].t_pulso[31] := 6000, d[0].t_pulso[32] := 6000, d[0].t_pulso[38] := 6000, d[0].precorte[2] := 1.0, d[0].precorte[3] := 1.0, d[0].precorte[4] := 1.0,
        d[0].precorte[5] := 1.0, d[0].precorte[6] := 0.5, d[0].precorte[7] := 0.5, d[0].precorte[8] := 0.5, d[0].precorte[9] := 0.5, d[0].precorte[10] := 1.0, d[0].precorte[11] := 1.0, d[0].precorte[12] := 1.0, d[0].precorte[13] := 1.0, d[0].precorte[14] := 0.5, d[0].precorte[15] := 0.5, d[0].precorte[16] := 0.5, d[0].precorte[17] := 0.5, d[0].precorte[18] := 0.1, d[0].precorte[19] := 0.1, d[0].precorte[20] := 0.1, d[0].precorte[21] := 0.1, d[0].precorte[22] := 0.1, d[0].precorte[23] := 0.1, d[0].precorte[24] := 0.1, d[0].precorte[26] := 0.1, d[0].precorte[27] := 0.1, d[0].precorte[28] := 0.1, d[0].precorte[29] := 0.1, d[0].precorte[30] := 0.1, d[0].precorte[31] := 0.1, d[0].precorte[32] := 0.1, d[0].precorte[38] := 0.1, d[0].error_per[2] := 5.0, d[0].error_per[3] := 5.0, d[0].error_per[4] := 5.0, d[0].error_per[5] := 5.0, d[0].error_per[6] := 5.0, d[0].error_per[7] := 5.0, d[0].error_per[8] := 5.0, d[0].error_per[9] := 5.0, d[0].error_per[10] := 5.0, d[0].error_per[11] := 5.0, d[0].error_per[12] := 5.0, d[0].error_per[13] := 5.0, d[0].error_per[14] := 5.0, d[0].error_per[15] := 5.0, d[0].error_per[16] := 5.0, d[0].error_per[17] := 5.0, d[0].error_per[18] := 5.0, d[0].error_per[19] := 5.0, d[0].error_per[20] := 5.0, d[0].error_per[21] := 5.0, d[0].error_per[22] := 5.0, d[0].error_per[23] := 5.0, d[0].error_per[24] := 5.0, d[0].error_per[25] := 5.0, d[0].error_per[26] := 5.0, d[0].error_per[27] := 5.0, d[0].error_per[28] := 5.0, d[0].error_per[29] := 5.0, d[0].error_per[30] := 5.0, d[0].error_per[31] := 5.0, d[0].error_per[32] := 5.0, d[0].error_per[38] := 5.0,
        d[0].error_kg[2] := 0.5, d[0].error_kg[3] := 0.5, d[0].error_kg[4] := 0.5, d[0].error_kg[5] := 0.5, d[0].error_kg[6] := 0.25, d[0].error_kg[7] := 0.25, d[0].error_kg[8] := 0.25, d[0].error_kg[9] := 0.25, d[0].error_kg[10] := 0.5, d[0].error_kg[11] := 0.5, d[0].error_kg[12] := 0.5, d[0].error_kg[13] := 0.5, d[0].error_kg[14] := 0.25, d[0].error_kg[15] := 0.25, d[0].error_kg[16] := 0.25, d[0].error_kg[17] := 0.25, d[0].error_kg[18] := 0.05, d[0].error_kg[19] := 0.05, d[0].error_kg[20] := 0.05, d[0].error_kg[21] := 0.05, d[0].error_kg[22] := 0.05, d[0].error_kg[23] := 0.05, d[0].error_kg[24] := 0.05, d[0].error_kg[25] := 0.25, d[0].error_kg[26] := 0.05, d[0].error_kg[27] := 0.05, d[0].error_kg[28] := 0.05, d[0].error_kg[29] := 0.05, d[0].error_kg[30] := 0.05, d[0].error_kg[31] := 0.05, d[0].error_kg[32] := 0.05, d[0].error_kg[38] := 0.25, d[0].frec_inicial[0] := 1.0, d[0].frec_inicial[2] := 50.0, d[0].frec_inicial[3] := 50.0, d[0].frec_inicial[4] := 50.0, d[0].frec_inicial[5] := 50.0, d[0].frec_inicial[6] := 50.0, d[0].frec_inicial[7] := 50.0, d[0].frec_inicial[8] := 50.0, d[0].frec_inicial[9] := 50.0, d[0].frec_inicial[10] := 50.0, d[0].frec_inicial[11] := 50.0, d[0].frec_inicial[12] := 50.0, d[0].frec_inicial[13] := 50.0, d[0].frec_inicial[14] := 50.0, d[0].frec_inicial[15] := 50.0, d[0].frec_inicial[16] := 50.0, d[0].frec_inicial[17] := 50.0, d[0].frec_inicial[18] := 50.0, d[0].frec_inicial[19] := 50.0, d[0].frec_inicial[20] := 50.0, d[0].frec_inicial[21] := 50.0, d[0].frec_inicial[22] := 50.0, d[0].frec_inicial[23] := 50.0, d[0].frec_inicial[24] := 50.0, d[0].frec_inicial[25] := 1.0, d[0].frec_inicial[26] := 50.0, d[0].frec_inicial[27] := 50.0, d[0].frec_inicial[28] := 50.0,
        d[0].frec_inicial[29] := 50.0, d[0].frec_inicial[30] := 50.0, d[0].frec_inicial[31] := 50.0, d[0].frec_inicial[32] := 50.0, d[0].frec_inicial[38] := 50.0, d[0].frec_final[0] := 1.0, d[0].frec_final[2] := 40.0, d[0].frec_final[3] := 40.0, d[0].frec_final[4] := 40.0, d[0].frec_final[5] := 40.0, d[0].frec_final[6] := 40.0, d[0].frec_final[7] := 40.0, d[0].frec_final[8] := 40.0, d[0].frec_final[9] := 40.0, d[0].frec_final[10] := 40.0, d[0].frec_final[11] := 40.0, d[0].frec_final[12] := 40.0, d[0].frec_final[13] := 40.0, d[0].frec_final[14] := 40.0, d[0].frec_final[15] := 40.0, d[0].frec_final[16] := 40.0, d[0].frec_final[17] := 40.0, d[0].frec_final[18] := 30.0, d[0].frec_final[19] := 30.0, d[0].frec_final[20] := 30.0, d[0].frec_final[21] := 30.0, d[0].frec_final[22] := 30.0, d[0].frec_final[23] := 30.0, d[0].frec_final[24] := 30.0, d[0].frec_final[25] := 1.0, d[0].frec_final[26] := 30.0, d[0].frec_final[27] := 30.0, d[0].frec_final[28] := 30.0, d[0].frec_final[29] := 30.0, d[0].frec_final[30] := 30.0, d[0].frec_final[31] := 30.0, d[0].frec_final[32] := 30.0, d[0].frec_final[38] := 40.0, d[0].curvatura[0] := 1.0, d[0].curvatura[2] := 4.0, d[0].curvatura[3] := 4.0, d[0].curvatura[4] := 4.0, d[0].curvatura[5] := 4.0, d[0].curvatura[6] := 3.0, d[0].curvatura[7] := 3.0, d[0].curvatura[8] := 3.0, d[0].curvatura[9] := 3.0, d[0].curvatura[10] := 4.0, d[0].curvatura[11] := 4.0, d[0].curvatura[12] := 4.0, d[0].curvatura[13] := 4.0, d[0].curvatura[14] := 3.0, d[0].curvatura[15] := 3.0, d[0].curvatura[16] := 3.0, d[0].curvatura[17] := 3.0, d[0].curvatura[18] := 1.0, d[0].curvatura[19] := 1.0, d[0].curvatura[20] := 1.0, d[0].curvatura[21] := 1.0, d[0].curvatura[22] := 1.0,
        d[0].curvatura[23] := 1.0, d[0].curvatura[24] := 1.0, d[0].curvatura[25] := 1.0, d[0].curvatura[26] := 1.0, d[0].curvatura[27] := 1.0, d[0].curvatura[28] := 1.0, d[0].curvatura[29] := 1.0, d[0].curvatura[30] := 1.0, d[0].curvatura[31] := 1.0, d[0].curvatura[32] := 1.0, d[0].curvatura[38] := 3.0, d[0].porcentaje_frec_max[0] := 1.0, d[0].porcentaje_frec_max[2] := 0.4, d[0].porcentaje_frec_max[3] := 0.4, d[0].porcentaje_frec_max[4] := 0.4, d[0].porcentaje_frec_max[5] := 0.4, d[0].porcentaje_frec_max[6] := 0.4, d[0].porcentaje_frec_max[7] := 0.4, d[0].porcentaje_frec_max[8] := 0.4, d[0].porcentaje_frec_max[9] := 0.4, d[0].porcentaje_frec_max[10] := 0.4, d[0].porcentaje_frec_max[11] := 0.4, d[0].porcentaje_frec_max[12] := 0.4, d[0].porcentaje_frec_max[13] := 0.4, d[0].porcentaje_frec_max[14] := 0.4, d[0].porcentaje_frec_max[15] := 0.4, d[0].porcentaje_frec_max[16] := 0.4, d[0].porcentaje_frec_max[17] := 0.4, d[0].porcentaje_frec_max[18] := 0.3, d[0].porcentaje_frec_max[19] := 0.3, d[0].porcentaje_frec_max[20] := 0.3, d[0].porcentaje_frec_max[21] := 0.3, d[0].porcentaje_frec_max[22] := 0.3, d[0].porcentaje_frec_max[23] := 0.3, d[0].porcentaje_frec_max[24] := 0.3, d[0].porcentaje_frec_max[25] := 1.0, d[0].porcentaje_frec_max[26] := 0.3, d[0].porcentaje_frec_max[27] := 0.3, d[0].porcentaje_frec_max[28] := 0.3, d[0].porcentaje_frec_max[29] := 0.3, d[0].porcentaje_frec_max[30] := 0.3, d[0].porcentaje_frec_max[31] := 0.3, d[0].porcentaje_frec_max[32] := 0.3, d[0].porcentaje_frec_max[38] := 0.4, d[0].high_limit[2] := 10.0, d[0].high_limit[3] := 10.0, d[0].high_limit[4] := 10.0, d[0].high_limit[5] := 10.0, d[0].high_limit[6] := 5.0, d[0].high_limit[7] := 5.0, d[0].high_limit[8] := 5.0, d[0].high_limit[9] := 5.0, d[0].high_limit[10] := 10.0, d[0].high_limit[11] := 10.0, d[0].high_limit[12] := 10.0, d[0].high_limit[13] := 10.0, d[0].high_limit[14] := 5.0, d[0].high_limit[15] := 5.0, d[0].high_limit[16] := 5.0, d[0].high_limit[17] := 5.0,
        d[0].high_limit[18] := 1.0, d[0].high_limit[19] := 1.0, d[0].high_limit[20] := 1.0, d[0].high_limit[21] := 1.0, d[0].high_limit[22] := 1.0, d[0].high_limit[23] := 1.0, d[0].high_limit[24] := 1.0, d[0].high_limit[25] := 5.0, d[0].high_limit[26] := 1.0, d[0].high_limit[27] := 1.0, d[0].high_limit[28] := 1.0, d[0].high_limit[29] := 1.0, d[0].high_limit[30] := 1.0, d[0].high_limit[31] := 1.0, d[0].high_limit[32] := 1.0, d[0].high_limit[38] := 1.0, d[1].t_espera[2] := 3000, d[1].t_espera[3] := 3000, d[1].t_espera[4] := 3000, d[1].t_espera[5] := 3000, d[1].t_espera[6] := 3000, d[1].t_espera[7] := 3000, d[1].t_espera[8] := 3000, d[1].t_espera[9] := 3000, d[1].t_espera[10] := 3000, d[1].t_espera[11] := 3000, d[1].t_espera[12] := 3000, d[1].t_espera[13] := 3000, d[1].t_espera[14] := 3000, d[1].t_espera[15] := 3000, d[1].t_espera[16] := 3000, d[1].t_espera[17] := 3000, d[1].t_espera[18] := 3000, d[1].t_espera[19] := 3000, d[1].t_espera[20] := 3000, d[1].t_espera[21] := 3000, d[1].t_espera[22] := 3000, d[1].t_espera[23] := 3000, d[1].t_espera[24] := 3000, d[1].t_espera[26] := 3000, d[1].t_espera[27] := 3000, d[1].t_espera[28] := 3000, d[1].t_espera[29] := 3000, d[1].t_espera[30] := 3000, d[1].t_espera[31] := 3000, d[1].t_espera[32] := 3000, d[1].t_espera[38] := 3000, d[1].t_pulso[2] := 10000, d[1].t_pulso[3] := 10000, d[1].t_pulso[4] := 10000, d[1].t_pulso[5] := 10000, d[1].t_pulso[6] := 10000, d[1].t_pulso[7] := 10000, d[1].t_pulso[8] := 10000, d[1].t_pulso[9] := 10000, d[1].t_pulso[10] := 10000, d[1].t_pulso[11] := 10000, d[1].t_pulso[12] := 10000, d[1].t_pulso[13] := 10000, d[1].t_pulso[14] := 10000,
        d[1].t_pulso[15] := 10000, d[1].t_pulso[16] := 10000, d[1].t_pulso[17] := 10000, d[1].t_pulso[18] := 6000, d[1].t_pulso[19] := 6000, d[1].t_pulso[20] := 6000, d[1].t_pulso[21] := 6000, d[1].t_pulso[22] := 6000, d[1].t_pulso[23] := 6000, d[1].t_pulso[24] := 6000, d[1].t_pulso[26] := 6000, d[1].t_pulso[27] := 6000, d[1].t_pulso[28] := 6000, d[1].t_pulso[29] := 6000, d[1].t_pulso[30] := 6000, d[1].t_pulso[31] := 6000, d[1].t_pulso[32] := 6000, d[1].t_pulso[38] := 6000, d[1].precorte[2] := 2.413803, d[1].precorte[3] := 1.8390074, d[1].precorte[4] := 2.1962054, d[1].precorte[5] := 3.0, d[1].precorte[6] := 0.86124694, d[1].precorte[7] := 1.297976, d[1].precorte[8] := 0.5, d[1].precorte[9] := 1.3912983, d[1].precorte[10] := 2.091219, d[1].precorte[11] := 3.0, d[1].precorte[12] := 2.2782488, d[1].precorte[13] := 3.0, d[1].precorte[14] := 1.3653834, d[1].precorte[15] := 1.102089, d[1].precorte[16] := 1.7, d[1].precorte[17] := 1.6370118, d[1].precorte[18] := 0.039811216, d[1].precorte[19] := 0.04979191, d[1].precorte[20] := 0.043874066, d[1].precorte[21] := 0.048747867, d[1].precorte[22] := 0.041324254, d[1].precorte[23] := 0.1, d[1].precorte[24] := 0.046323393, d[1].precorte[26] := 0.049721815, d[1].precorte[27] := 0.025162328, d[1].precorte[28] := 0.052942604, d[1].precorte[29] := 0.05468315, d[1].precorte[30] := 0.1, d[1].precorte[31] := 0.050990697, d[1].precorte[32] := 0.1, d[1].precorte[38] := 0.2662258, d[1].error_per[2] := 5.0, d[1].error_per[3] := 5.0, d[1].error_per[4] := 5.0, d[1].error_per[5] := 5.0, d[1].error_per[6] := 5.0, d[1].error_per[7] := 5.0, d[1].error_per[8] := 5.0, d[1].error_per[9] := 5.0, d[1].error_per[10] := 5.0, d[1].error_per[11] := 5.0, d[1].error_per[12] := 5.0,
        d[1].error_per[13] := 5.0, d[1].error_per[14] := 5.0, d[1].error_per[15] := 5.0, d[1].error_per[16] := 5.0, d[1].error_per[17] := 5.0, d[1].error_per[18] := 5.0, d[1].error_per[19] := 5.0, d[1].error_per[20] := 5.0, d[1].error_per[21] := 5.0, d[1].error_per[22] := 5.0, d[1].error_per[23] := 5.0, d[1].error_per[24] := 5.0, d[1].error_per[25] := 5.0, d[1].error_per[26] := 5.0, d[1].error_per[27] := 5.0, d[1].error_per[28] := 5.0, d[1].error_per[29] := 5.0, d[1].error_per[30] := 5.0, d[1].error_per[31] := 5.0, d[1].error_per[32] := 5.0, d[1].error_per[38] := 5.0, d[1].error_kg[2] := 5.0, d[1].error_kg[3] := 5.0, d[1].error_kg[4] := 5.0, d[1].error_kg[5] := 5.0, d[1].error_kg[6] := 0.5, d[1].error_kg[7] := 0.5, d[1].error_kg[8] := 0.5, d[1].error_kg[9] := 0.5, d[1].error_kg[10] := 5.0, d[1].error_kg[11] := 5.0, d[1].error_kg[12] := 5.0, d[1].error_kg[13] := 5.0, d[1].error_kg[14] := 0.5, d[1].error_kg[15] := 0.5, d[1].error_kg[16] := 0.5, d[1].error_kg[17] := 0.5, d[1].error_kg[18] := 0.1, d[1].error_kg[19] := 0.1, d[1].error_kg[20] := 0.1, d[1].error_kg[21] := 0.1, d[1].error_kg[22] := 0.1, d[1].error_kg[23] := 0.1, d[1].error_kg[24] := 0.1, d[1].error_kg[25] := 0.5, d[1].error_kg[26] := 0.1, d[1].error_kg[27] := 0.1, d[1].error_kg[28] := 0.1, d[1].error_kg[29] := 0.1, d[1].error_kg[30] := 0.1, d[1].error_kg[31] := 0.1, d[1].error_kg[32] := 0.1, d[1].error_kg[38] := 0.5, d[1].frec_inicial[0] := 1.0, d[1].frec_inicial[2] := 70.0, d[1].frec_inicial[3] := 70.0, d[1].frec_inicial[4] := 70.0, d[1].frec_inicial[5] := 70.0, d[1].frec_inicial[6] := 70.0, d[1].frec_inicial[7] := 70.0,
        d[1].frec_inicial[8] := 70.0, d[1].frec_inicial[9] := 70.0, d[1].frec_inicial[10] := 70.0, d[1].frec_inicial[11] := 70.0, d[1].frec_inicial[12] := 70.0, d[1].frec_inicial[13] := 70.0, d[1].frec_inicial[14] := 70.0, d[1].frec_inicial[15] := 70.0, d[1].frec_inicial[16] := 70.0, d[1].frec_inicial[17] := 70.0, d[1].frec_inicial[18] := 70.0, d[1].frec_inicial[19] := 70.0, d[1].frec_inicial[20] := 70.0, d[1].frec_inicial[21] := 70.0, d[1].frec_inicial[22] := 70.0, d[1].frec_inicial[23] := 70.0, d[1].frec_inicial[24] := 70.0, d[1].frec_inicial[25] := 1.0, d[1].frec_inicial[26] := 70.0, d[1].frec_inicial[27] := 70.0, d[1].frec_inicial[28] := 70.0, d[1].frec_inicial[29] := 70.0, d[1].frec_inicial[30] := 70.0, d[1].frec_inicial[31] := 70.0, d[1].frec_inicial[32] := 70.0, d[1].frec_inicial[38] := 50.0, d[1].frec_final[0] := 1.0, d[1].frec_final[2] := 50.0, d[1].frec_final[3] := 50.0, d[1].frec_final[4] := 50.0, d[1].frec_final[5] := 50.0, d[1].frec_final[6] := 50.0, d[1].frec_final[7] := 50.0, d[1].frec_final[8] := 50.0, d[1].frec_final[9] := 50.0, d[1].frec_final[10] := 50.0, d[1].frec_final[11] := 50.0, d[1].frec_final[12] := 50.0, d[1].frec_final[13] := 50.0, d[1].frec_final[14] := 50.0, d[1].frec_final[15] := 50.0, d[1].frec_final[16] := 50.0, d[1].frec_final[17] := 50.0, d[1].frec_final[18] := 50.0, d[1].frec_final[19] := 50.0, d[1].frec_final[20] := 50.0, d[1].frec_final[21] := 50.0, d[1].frec_final[22] := 50.0, d[1].frec_final[23] := 50.0, d[1].frec_final[24] := 50.0, d[1].frec_final[25] := 1.0, d[1].frec_final[26] := 50.0, d[1].frec_final[27] := 50.0, d[1].frec_final[28] := 50.0, d[1].frec_final[29] := 50.0, d[1].frec_final[30] := 50.0, d[1].frec_final[31] := 50.0, d[1].frec_final[32] := 50.0, d[1].frec_final[38] := 40.0, d[1].curvatura[0] := 1.0,
        d[1].curvatura[2] := 4.0, d[1].curvatura[3] := 4.0, d[1].curvatura[4] := 4.0, d[1].curvatura[5] := 4.0, d[1].curvatura[6] := 3.0, d[1].curvatura[7] := 3.0, d[1].curvatura[8] := 3.0, d[1].curvatura[9] := 3.0, d[1].curvatura[10] := 4.0, d[1].curvatura[11] := 4.0, d[1].curvatura[12] := 4.0, d[1].curvatura[13] := 4.0, d[1].curvatura[14] := 3.0, d[1].curvatura[15] := 3.0, d[1].curvatura[16] := 3.0, d[1].curvatura[17] := 3.0, d[1].curvatura[18] := 1.0, d[1].curvatura[19] := 1.0, d[1].curvatura[20] := 1.0, d[1].curvatura[21] := 1.0, d[1].curvatura[22] := 1.0, d[1].curvatura[23] := 1.0, d[1].curvatura[24] := 1.0, d[1].curvatura[25] := 1.0, d[1].curvatura[26] := 1.0, d[1].curvatura[27] := 1.0, d[1].curvatura[28] := 1.0, d[1].curvatura[29] := 1.0, d[1].curvatura[30] := 1.0, d[1].curvatura[31] := 1.0, d[1].curvatura[32] := 1.0, d[1].curvatura[38] := 3.0, d[1].porcentaje_frec_max[0] := 1.0, d[1].porcentaje_frec_max[2] := 0.6, d[1].porcentaje_frec_max[3] := 0.6, d[1].porcentaje_frec_max[4] := 0.6, d[1].porcentaje_frec_max[5] := 0.6, d[1].porcentaje_frec_max[6] := 0.6, d[1].porcentaje_frec_max[7] := 0.6, d[1].porcentaje_frec_max[8] := 0.6, d[1].porcentaje_frec_max[9] := 0.6, d[1].porcentaje_frec_max[10] := 0.6, d[1].porcentaje_frec_max[11] := 0.6, d[1].porcentaje_frec_max[12] := 0.6, d[1].porcentaje_frec_max[13] := 0.6, d[1].porcentaje_frec_max[14] := 0.6, d[1].porcentaje_frec_max[15] := 0.6, d[1].porcentaje_frec_max[16] := 0.6, d[1].porcentaje_frec_max[17] := 0.6, d[1].porcentaje_frec_max[18] := 0.5, d[1].porcentaje_frec_max[19] := 0.5, d[1].porcentaje_frec_max[20] := 0.5, d[1].porcentaje_frec_max[21] := 0.5, d[1].porcentaje_frec_max[22] := 0.5, d[1].porcentaje_frec_max[23] := 0.5, d[1].porcentaje_frec_max[24] := 0.5, d[1].porcentaje_frec_max[25] := 1.0, d[1].porcentaje_frec_max[26] := 0.5, d[1].porcentaje_frec_max[27] := 0.5, d[1].porcentaje_frec_max[28] := 0.5,
        d[1].porcentaje_frec_max[29] := 0.5, d[1].porcentaje_frec_max[30] := 0.5, d[1].porcentaje_frec_max[31] := 0.5, d[1].porcentaje_frec_max[32] := 0.5, d[1].porcentaje_frec_max[38] := 0.5, d[1].low_limit[2] := 10.0, d[1].low_limit[3] := 10.0, d[1].low_limit[4] := 10.0, d[1].low_limit[5] := 10.0, d[1].low_limit[6] := 5.0, d[1].low_limit[7] := 5.0, d[1].low_limit[8] := 5.0, d[1].low_limit[9] := 5.0, d[1].low_limit[10] := 10.0, d[1].low_limit[11] := 10.0, d[1].low_limit[12] := 10.0, d[1].low_limit[13] := 10.0, d[1].low_limit[14] := 5.0, d[1].low_limit[15] := 5.0, d[1].low_limit[16] := 5.0, d[1].low_limit[17] := 5.0, d[1].low_limit[18] := 1.0, d[1].low_limit[19] := 1.0, d[1].low_limit[20] := 1.0, d[1].low_limit[21] := 1.0, d[1].low_limit[22] := 1.0, d[1].low_limit[23] := 1.0, d[1].low_limit[24] := 1.0, d[1].low_limit[25] := 5.0, d[1].low_limit[26] := 1.0, d[1].low_limit[27] := 1.0, d[1].low_limit[28] := 1.0, d[1].low_limit[29] := 1.0, d[1].low_limit[30] := 1.0, d[1].low_limit[31] := 1.0, d[1].low_limit[32] := 1.0, d[1].low_limit[38] := 1.0, d[1].high_limit[2] := 999999.0, d[1].high_limit[3] := 999999.0, d[1].high_limit[4] := 999999.0, d[1].high_limit[5] := 999999.0, d[1].high_limit[6] := 999999.0, d[1].high_limit[7] := 999999.0, d[1].high_limit[8] := 999999.0, d[1].high_limit[9] := 999999.0, d[1].high_limit[10] := 999999.0, d[1].high_limit[11] := 999999.0, d[1].high_limit[12] := 999999.0, d[1].high_limit[13] := 999999.0, d[1].high_limit[14] := 999999.0, d[1].high_limit[15] := 999999.0, d[1].high_limit[16] := 999999.0, d[1].high_limit[17] := 999999.0, d[1].high_limit[18] := 999999.0, d[1].high_limit[19] := 999999.0, d[1].high_limit[20] := 999999.0, d[1].high_limit[21] := 999999.0, d[1].high_limit[22] := 999999.0, d[1].high_limit[23] := 999999.0, d[1].high_limit[24] := 999999.0,
        d[1].high_limit[25] := 999999.0, d[1].high_limit[26] := 999999.0, d[1].high_limit[27] := 999999.0, d[1].high_limit[28] := 999999.0, d[1].high_limit[29] := 999999.0, d[1].high_limit[30] := 999999.0, d[1].high_limit[31] := 999999.0, d[1].high_limit[32] := 999999.0, d[1].high_limit[38] := 999999.0);
        [0]   // Pequeño
        [1]   // Grande
   TabDosif : tabDosif := (idx_tolva[0] := 33, idx_tolva[1] := 34, idx_tolva[2] := 35, idx_tolva[3] := 36, idx_tolva[4] := 25, idx_tolva[5] := 38, idx_vdf[0] := 1, idx_vdf[1] := 2, idx_vdf[2] := 3, idx_vdf[3] := 4, idx_vdf[5] := 5);
   Timer : TIMER[500] := ([0].PRE := 2000, [0].ACC := 1000, [1].PRE := 60000, [2].PRE := 60000, [3].PRE := 60000, [4].PRE := 60000, [5].PRE := 60000, [6].PRE := 50000, [7].PRE := 60000, [8].PRE := 3000, [8].ACC := 117, [8].EN := 1, [8].TT := 1, [9].PRE := 8000, [9].ACC := 1558, [9].EN := 1, [9].TT := 1, [10].PRE := 5000, [11].PRE := 3501, [12].PRE := 3000, [13].PRE := 3000, [14].PRE := 1100, [15].PRE := 1100, [16].PRE := 300000, [17].PRE := 3000, [18].PRE := 3000, [19].PRE := 5000, [20].PRE := 2000, [21].PRE := 3000, [22].PRE := 3000, [23].PRE := 2000, [24].PRE := 3000, [25].PRE := 2000, [26].PRE := 5000, [27].PRE := 3000, [28].PRE := 2000, [29].PRE := 3000, [30].PRE := 20000, [31].PRE := 20000, [32].PRE := 10000, [33].PRE := 10000, [34].PRE := 30000, [35].PRE := 5000, [36].PRE := 10000, [37].PRE := 10000, [38].PRE := 10000, [39].PRE := 4000, [40].PRE := 60000, [41].PRE := 7000, [42].PRE := 3000, [43].PRE := 10000, [44].PRE := 10000, [45].PRE := 2000, [46].PRE := 3000, [47].PRE := 60000, [48].PRE := 5000, [49].PRE := 20000, [50].PRE := 1000, [50].ACC := 962, [50].EN := 1,
        [50].TT := 1, [51].PRE := 1000, [51].ACC := 962, [51].EN := 1, [51].TT := 1, [52].PRE := 1000, [52].ACC := 962, [52].EN := 1, [52].TT := 1, [53].PRE := 1000, [53].ACC := 962, [53].EN := 1, [53].TT := 1, [54].PRE := 3000, [55].PRE := 3000, [55].ACC := 2058, [55].EN := 1, [55].TT := 1, [56].PRE := 3000, [57].PRE := 2000, [58].PRE := 10000, [59].PRE := 10000, [60].PRE := 10000, [61].PRE := 30000, [62].PRE := 3000, [63].PRE := 30000, [64].PRE := 10000, [65].PRE := 5000, [66].PRE := 60000, [67].PRE := 10000, [68].PRE := 3000, [69].PRE := 10000, [70].PRE := 30000, [71].PRE := 3000, [72].PRE := 20000, [73].PRE := 10000, [74].PRE := 10000, [75].PRE := 10000, [76].PRE := 10000, [77].PRE := 5000, [78].PRE := 2000, [79].PRE := 2000, [80].PRE := 5000, [81].PRE := 5000, [82].PRE := 5000, [83].PRE := 5000, [84].PRE := 10000, [85].PRE := 5000, [86].PRE := 5000, [87].PRE := 5000, [88].PRE := 5000, [89].PRE := 5000, [90].PRE := 5000, [91].PRE := 5000, [92].PRE := 5000, [93].PRE := 5000, [94].PRE := 5000, [95].PRE := 5000, [96].PRE := 5000, [97].PRE := 5000,
        [97].EN := 1, [97].TT := 1, [98].PRE := 5000, [99].PRE := 5000, [100].PRE := 900000, [101].PRE := 5000, [102].PRE := 600000, [103].PRE := 3000, [104].PRE := 5000, [105].PRE := 5000, [106].PRE := 5000, [107].PRE := 5000, [108].PRE := 5000, [109].PRE := 5000, [110].PRE := 2000, [110].ACC := 1327, [110].EN := 1, [110].TT := 1, [111].PRE := 5000, [112].PRE := 600000, [113].PRE := 3000, [114].PRE := 5000, [115].PRE := 5000, [116].PRE := 5000, [117].PRE := 30000, [118].PRE := 30000, [119].PRE := 60000, [120].PRE := 500, [121].PRE := 200, [121].ACC := 142, [121].EN := 1, [121].TT := 1, [122].PRE := 5000, [123].PRE := 3000, [124].PRE := 2000, [125].PRE := 3000, [126].PRE := 2000, [127].PRE := 3000, [128].PRE := 2000, [130].PRE := 30000, [131].PRE := 30000, [132].PRE := 30000, [133].PRE := 30000, [134].PRE := 5000, [135].PRE := 300000, [136].PRE := 300000, [137].PRE := 30000, [140].PRE := 16, [141].PRE := 4, [142].PRE := 2000, [143].PRE := 2000, [144].PRE := 5000, [145].PRE := 5000, [146].PRE := 10000, [147].PRE := 30000, [148].PRE := 10000, [149].PRE := 30000, [150].PRE := 120000, [151].PRE := 120000, [152].PRE := 10000,
        [152].ACC := 10085, [153].PRE := 10000, [153].ACC := 10087, [154].PRE := 3000, [155].PRE := 3000, [156].PRE := 5000, [157].PRE := 1000, [158].PRE := 5000, [159].PRE := 15000, [160].PRE := 3000, [161].PRE := 2650, [162].PRE := 10000, [163].PRE := 60000, [164].PRE := 10000, [165].PRE := 60000, [166].PRE := 10000, [167].PRE := 30000, [168].PRE := 7500, [169].PRE := 30000, [170].PRE := 5000, [171].PRE := 5000, [172].PRE := 5000, [173].PRE := 5000, [174].PRE := 5000, [175].PRE := 5000, [176].PRE := 60000, [177].PRE := 60000, [178].PRE := 3000, [178].ACC := 366, [178].EN := 1, [178].TT := 1, [179].PRE := 1000, [180].PRE := 60000, [181].PRE := 60000, [182].PRE := 2000, [182].ACC := 2039, [183].PRE := 3000, [183].ACC := 3000, [184].PRE := 3000, [185].PRE := 1500000, [185].ACC := 1500000, [186].PRE := 10000, [186].ACC := 9757, [186].EN := 1, [186].TT := 1, [187].PRE := 3000, [190].PRE := 1000, [190].ACC := 1061, [190].EN := 1, [190].DN := 1, [191].PRE := 1000, [191].ACC := 1061, [191].EN := 1, [191].DN := 1, [192].PRE := 5000, [193].PRE := 2000, [194].PRE := 2000, [195].PRE := 2000, [196].PRE := 60000, [197].PRE := 2000,
        [198].PRE := 3000, [199].PRE := 3000, [200].PRE := 2000, [201].PRE := 3000, [202].PRE := 5000, [203].PRE := 3000, [203].ACC := 273, [204].PRE := 3000, [204].ACC := 560, [204].EN := 1, [204].TT := 1, [205].PRE := 3000, [206].PRE := 5000, [207].PRE := 2000, [208].PRE := 50000, [209].PRE := 500, [210].PRE := 2000, [211].PRE := 5000, [212].PRE := 1000, [213].PRE := 3000, [214].PRE := 2000, [215].PRE := 3000, [216].PRE := 1000, [217].PRE := 3000, [218].PRE := 2000, [219].PRE := 3000, [220].PRE := 5000, [221].PRE := 3000, [222].PRE := 3000, [224].PRE := 5000, [225].PRE := 10000, [230].PRE := 2000, [231].PRE := 3000, [240].PRE := 2000, [241].PRE := 3000, [242].PRE := 30000, [243].PRE := 180000, [244].PRE := 3000, [245].PRE := 300000, [246].PRE := 30000, [247].PRE := 180000, [248].PRE := 3000, [249].PRE := 120000, [250].PRE := 3000, [250].ACC := 280, [250].EN := 1, [250].TT := 1, [251].PRE := 3000, [252].PRE := 5000, [253].PRE := 2000, [260].PRE := 2000, [261].PRE := 6000, [270].PRE := 3000, [271].PRE := 5000, [271].ACC := 3078, [271].EN := 1, [271].TT := 1, [272].PRE := 1000, [273].PRE := 1000, [273].ACC := 1026,
        [273].EN := 1, [273].DN := 1, [300].PRE := 1000, [301].PRE := 5000, [302].PRE := 1000, [303].PRE := 5000, [350].PRE := 3000, [350].ACC := 720, [350].EN := 1, [350].TT := 1, [351].PRE := 3000, [351].ACC := 720, [351].EN := 1, [351].TT := 1, [352].PRE := 3000, [352].ACC := 360, [352].EN := 1, [352].TT := 1, [353].PRE := 3000, [353].EN := 1, [353].TT := 1, [354].PRE := 3000, [354].ACC := 2160, [354].EN := 1, [354].TT := 1, [355].PRE := 10000, [355].ACC := 9010, [355].EN := 1, [355].TT := 1, [400].PRE := 1000, [400].EN := 1, [400].TT := 1, [401].PRE := 3000, [401].EN := 1, [401].DN := 1, [402].PRE := 500, [402].EN := 1, [402].TT := 1, [410].PRE := 3000, [411].PRE := 3000, [411].ACC := 3000, [412].PRE := 100, [420].PRE := 3000, [421].PRE := 3000, [421].ACC := 3000, [422].PRE := 100, [423].PRE := 60000, [430].PRE := 3000, [431].PRE := 3000, [431].ACC := 3000, [432].PRE := 100, [440].PRE := 3000, [441].PRE := 3000, [441].ACC := 3000, [442].PRE := 100, [446].PRE := 10000, [446].ACC := 7100, [446].EN := 1, [446].TT := 1, [450].PRE := 3000,
        [451].PRE := 3000, [451].ACC := 3000, [452].PRE := 100, [460].PRE := 3000, [461].PRE := 3000, [461].ACC := 3000, [462].PRE := 100, [470].PRE := 5000, [471].PRE := 5000, [472].PRE := 20000, [473].PRE := 20000, [474].PRE := 20000, [475].PRE := 20000, [476].PRE := 20000, [477].PRE := 20000, [478].PRE := 30000, [479].PRE := 200000, [480].PRE := 60000, [480].ACC := 60883, [480].EN := 1, [480].DN := 1, [481].PRE := 5000, [482].PRE := 30000, [483].PRE := 20000, [484].PRE := 10000, [485].PRE := 60000, [486].PRE := 20000, [487].PRE := 20000, [488].PRE := 20000, [489].PRE := 200000, [490].PRE := 20000, [491].PRE := 30000, [492].PRE := 30000, [493].PRE := 10000, [494].PRE := 5000, [495].PRE := 5000, [496].PRE := 5000, [497].PRE := 180000);
        [17]   // Timer retardo refresco de datos antes de trigger
        [8]   // Timer Wdog
        [9]   // Timer Retry Wdog
        [10]   // Tpo Esp Antes Trigger WD
        [204]   // Trigger Waits Data Refresh
        [210]   // Tpo entre pedidos
        [213]   // Timeout req line
   Value : DINT[500] := ([0] := 2014, [1] := 5, [2] := 15, [3] := 18, [4] := 46, [5] := 46, [6] := 633015, [8] := 18032565, [10] := 127, [11] := 5017, [12] := 45, [13] := 2, [15] := 2063468288, [18] := 11544539, [22] := 4, [23] := 10, [25] := 12, [26] := 3, [28] := 5, [29] := 59, [30] := 1, [31] := 1, [33] := 1, [34] := 1, [35] := 3, [36] := 1, [37] := 1332, [38] := 1, [41] := 461, [49] := 210, [50] := 10, [51] := 1, [52] := 65, [53] := 1074237440, [55] := 43, [57] := 2, [62] := 65, [63] := 497664, [64] := 5226, [65] := 125022003, [67] := 2, [72] := 81, [73] := 2600960, [74] := 5, [75] := 100, [77] := 2, [79] := 10, [82] := 689, [87] := 4, [92] := 2478, [93] := 53793, [94] := 2521, [95] := 1, [99] := 2103, [100] := 1, [101] := 1, [103] := 1, [104] := 4, [105] := 500, [108] := 1579,
        [109] := -575, [113] := 1, [114] := 4, [115] := 1579, [122] := 81, [123] := 2600960, [124] := 16, [125] := 17, [126] := 112, [127] := 123, [131] := 24578, [132] := 2, [135] := 6, [137] := 1, [142] := -8189, [143] := -8189, [144] := 559, [147] := 16, [151] := 11, [153] := 22, [155] := 11, [157] := 1, [161] := 1, [163] := 44, [167] := 1, [169] := 1, [171] := 1, [173] := 1, [175] := 1, [177] := 1, [179] := 1, [201] := 1, [202] := 1, [203] := 1, [204] := 1, [205] := 1, [206] := 1, [207] := 1, [208] := 1, [209] := 1, [212] := 1, [214] := 2, [216] := 18, [217] := 20573367, [218] := 20573367, [219] := 99, [220] := 20574109, [221] := 20574109, [222] := 2, [223] := 18, [224] := 99, [225] := 18, [226] := -1, [227] := 99, [228] := 2, [229] := 2, [230] := 20070515, [231] := 19183654, [233] := 19183654, [234] := 7,
        [235] := 10, [236] := 1, [237] := 20070720, [238] := 18582492, [239] := 100, [240] := 18582492, [241] := 2303, [242] := 3, [243] := 1, [252] := 3, [253] := 1, [254] := 3, [255] := 1, [257] := 1519, [258] := 19443816, [261] := 255, [262] := 100, [264] := 1, [273] := 255, [274] := 100, [282] := 805306378, [284] := 56, [285] := 50, [287] := 50, [290] := 14, [293] := -1, [294] := 15, [295] := 15, [298] := 110, [299] := 8, [300] := 108, [301] := 761299, [302] := 133, [303] := 1, [307] := 5, [308] := 2, [310] := 2133, [312] := 1, [313] := 114, [314] := 32, [317] := 1, [319] := 14, [320] := 100, [321] := 7, [322] := 6969, [323] := 618, [324] := 3, [327] := 98, [329] := 2, [330] := 4, [331] := 2, [332] := 7, [333] := 1, [336] := 86, [339] := 77, [340] := 777, [341] := 1, [342] := 7777, [343] := 107, [344] := 6,
        [347] := 99, [349] := 14, [360] := 123456789, [361] := 1, [362] := 111, [363] := 420, [364] := 14, [367] := 98, [370] := 223, [371] := 1, [372] := 2312, [373] := 15, [374] := 15, [377] := 99, [380] := 223, [381] := 1, [382] := 2312, [383] := 15, [384] := 5, [385] := 6, [386] := 8, [387] := 100, [398] := 134217727, [405] := 6, [406] := 20070714, [407] := 20255021, [408] := 1, [410] := 123456789, [411] := 1, [412] := 111, [413] := 420, [414] := 14, [419] := 6, [420] := 223, [421] := 1, [422] := 2312, [423] := 15, [424] := 15, [428] := 3, [429] := 6, [450] := -1, [461] := 3, [465] := 4, [498] := 255, [499] := 3);
        [18].23   // Selector Man(0)/Auto(1) TDF_101
        [159]   // Password Interfaz 5 (Disponible)
        [161]   // Password Interfaz 6 (HMI Intake)
        [15].1   // Recepción automatica de batch
        [150]   // Usuario Interfaz 1 (PanelView #1)
        [323]   // Pop intake PanelView 1 - Cod_MP
        [152]   // Usuario Interfaz 2 (PanelView #2)
        [358]   // Comando PV4
        [154]   // Usuario Interfaz 3 (PanelView #3)
        [400]   // Num Guia Termino mov MP
        [401]   // Item Guia Termino mov MP
        [402]   // Usuario Termino mov MP
        [15].12   // Aviso descarga previa Micros
        [15].13   // Ejecutar desc. Previa Micros
        [26].1   // Login Interfaz 1
        [26].2   // Login Interfaz 2
        [26].6   // Login Interfaz 6
        [26].7   // Login Interfaz 7
        [26].15   // Login Interfaz #01
        [403]   // Codigo MP Termino mov MP
        [405]   // Interfaz Termino mov MP
        [156]   // Usuario Interfaz 4 (PanelView #4)
        [406]   // Fecha Termino mov MP
        [407]   // Timestamp Termino mov MP
        [408]   // Tipo Termino (1) Auto (2) Man
        [168]   // Usuario Interfaz 10 (HMI ServAux)
        [409]   // Cod Error mov MP
        [425]   // Actual en Ruta 2 - Bin B
        [242]   // Usuario Interfaz 1 (PanelView #1)
        [460]   // Resultado Macro1
        [460].0   // Flag Fuera de Tolva
        [461]   // Índice de Ingrediente Mac1
        [462]   // Mensajes Mac1
        [244]   // Usuario Interfaz 2 (PanelView #2)
        [463]   // Respuestas Mac1
        [464]   // Resultado Macro2
        [246]   // Usuario Interfaz 3 (PanelView #3)
        [465]   // Índice de Ingrediente Mac2
        [466]   // Mensajes Mac2
        [248]   // Usuario Interfaz 4 (PanelView #4)
        [467]   // Respuestas Mac2
        [468]   // Resultado Midi
        [469]   // Índice de Ingredientes Midi
        [470]   // Mensajes Midi
        [471]   // Respuestas Midi
        [472]   // Resultado Micro
        [473]   // Índice de Ingredientes Micro
        [474]   // Mensajes Micro
        [475]   // Respuestas Micro
        [476]   // Resultado Liq1
        [477]   // Índice de Ingrediente Liq1
        [478]   // Mensajes Liq1
        [479]   // Respuestas Liq1
        [480]   // Resultado Liq2
        [481]   // Índice de Ingrediente Liq2
        [482]   // Mensajes Liq2
        [483]   // Respuestas Liq2
        [484]   // Resultado Liq3
        [485]   // Índice de Ingrediente Liq3
        [486]   // Mensajes Liq3
        [311]   // Tipo Termino Ruta 1 Automático (=1) Manual (=0)
        [26].16   // Login Interfaz #02
        [487]   // Respuestas Liq3
        [488]   // Resultado Liq4
        [26].17   // Login Interfaz #03
        [26].18   // Login Interfaz #04
        [489]   // Índice de Ingrediente Liq4
        [490]   // Mensajes Liq4
        [491]   // Respuestas Liq4
        [492]   // Resultado Liq5
        [493]   // Índice de Ingrediente Liq5
        [494]   // Mensajes Liq5
        [495]   // Respuestas Liq5
        [26].19   // Login Interfaz #05
        [26].20   // Login Interfaz #06
        [26].21   // Login Interfaz #07
        [312]   // Tipo Termino Ruta 2 Automático (=1) Manual (=0)
        [26].22   // Login Interfaz #08
        [26].23   // Login Interfaz #09
        [26].24   // Login Interfaz #10
        [261]   // Nivel de Acceso Interfaz 1 (PanelView #1)
        [26].25   // Login Interfaz #11
        [27].15   // Login Interfaz 1
        [28].0   // Error Comm Buffer mov MP
        [28].1   // Error Comm ReportDMM DMM
        [28].3   // Error Comm Import MP
        [28].4   // Bin Reproceso Vacío
        [29].0   // RSSql Timeout
        [29].1   // Error Comm con DMM
        [29].2   // Bitacora Llena
        [320]   // Pop intake PanelView 1 - Numero de Guia
        [29].3   // Error Comm en Bitácora
        [263]   // Nivel de Acceso Interfaz 2 (PanelView #2)
        [265]   // Nivel de Acceso Interfaz 3 (PanelView #3)
        [322]   // Pop intake PanelView 1 - Patente Camión
        [267]   // Nivel de Acceso Interfaz 4 (PanelView #4)
        [371]   // Pop intake Ruta 2 PC Intake - Item Guia
        [29].4   // Error Comm en ID Batch
        [29].5   // Error Comm Report Batch
        [377]   // Transmisión Input MP Ruta 2 PC Intake - Cod_Error
        [29].10   // SurgeBin Refill L1
        [29].11   // SurgeBin Refill L2
        [39]   // Tiempo Real Dosificación Macros
        [40]   // Tpo Efectivo Micros
        [41].1   // Intake Cmd Ok Login
        [7].17   // Destination Mode Without Barcode
        [43]   // Tiempo Real Premezclado Linea#1
        [44]   // Tiempo Mezclado Linea#1
        [45]   // Tiempo Real Premezclado Linea#2
        [46]   // Tiempo hacia LiveBin #3
        [47]   // Tpo Transporte LiveBin L1
        [48]   // Tpo Transporte LiveBin L2
        [50]   // RSV Index AB_Abajo
        [42]   // Tiempo Real Transporte hacia Lineas
        [51]   // Index_Old AB Abajo
        [151]   // Password Interfaz 1 (PanelView #1)
        [52]   // Out D Direct
        [56]   // RSV Cmd AB_Abajo
        [262]   // Cod. Error Interfaz 1 (PanelView #1)
        [153]   // Password Interfaz 2 (PanelView #2)
        [155]   // Password Interfaz 3 (PanelView #3)
        [157]   // Password Interfaz 4 (PanelView #4)
        [243]   // Password Interfaz 1 (PanelView #1)
        [245]   // Password Interfaz 2 (PanelView #2)
        [309]   // Con (=1), sin (=0) Conexión a BD Guías
        [247]   // Password Interfaz 3 (PanelView #3)
        [249]   // Password Interfaz 4 (PanelView #4)
        [272]   // Cod. Error Interfaz 6 (HMI Intake)
        [289]   // Common PID Popup Window - Commands
        [100].10   // _
        [158]   // Usuario Interfaz 5 (Disponible)
        [160]   // Usuario Interfaz 6 (HMI Intake)
        [327]   // Transmisión Input MP PanelView 1 - Cod_Error
        [264]   // Cod. Error Interfaz 2 (PanelView #2)
        [100].11   // _
        [100].12   // _
        [100].13   // _
        [100].14   // _
        [100].15   // _
        [100].16   // _
        [100].17   // _
        [252]   // Usuario Interfaz 6 (HMI Intake)
        [100].18   // _
        [100].19   // _
        [266]   // Cod. Error Interfaz 3 (PanelView #3)
        [268]   // Cod. Error Interfaz 4 (PanelView #4)
        [368]   // Comando desde Terminal (Revisar=1, SetRuta=2) Ruta 1 PC Intake
        [100].20   // _
        [274]   // Cod. Error Interfaz 7 (HMI DMM)
        [271]   // Nivel de Acceso Interfaz 6 (HMI Intake)
        [281]   // PID Index from RSView - old
        [100].21   // _
        [100].22   // _
        [344]   // Total Production since recipe Change
        [373]   // Pop intake Ruta 2 PC Intake - Cod_MP
        [100].23   // _
        [283]   // Common PID Popup Window - PV
        [100].24   // _
        [100].25   // _
        [100].26   // _
        [378]   // Comando desde Terminal (Revisar=1, SetRuta=2) Ruta 2 PC Intake
        [100].27   // _
        [284]   // Common PID Popup Window - SP
        [273]   // Nivel de Acceso Interfaz 7 (HMI DMM)
        [285]   // Common PID Popup Window - CV
        [282]   // Common PID Popup Window Status Bits1
        [374]   // Pop intake Ruta 2 PC Intake - Bin A
        [101].10   // _
        [286]   // Common PID Popup Window - AI
        [375]   // Pop intake Ruta 2 PC Intake - Bin B
        [101].11   // _
        [287]   // Common PID Popup Window - AO
        [102].10   // _
        [293]   // Eqp Tolva Destino Ruta 1
        [18].13   // "Selector Man(0)/Auto(1) TDF_082 y TDF_085"
        [102].11   // _
        [376]   // Pop intake Ruta 2 PC Intake - Bin C
        [370]   // Pop intake Ruta 2 PC Intake - Numero de Guia
        [372]   // Pop intake Ruta 2 PC Intake - Patente Camión
        [294]   // Indice dentro Origen Ruta 1
        [102].12   // _
        [102].13   // _
        [102].14   // _
        [297]   // Codigo de Error
        [7].16   // Destination Mode With Barcode Automatic
        [308]   // Comando Revisar(=1) o Set_Ruta(=2) PC Intake
        [298]   // Eqp Tolva Destino Ruta 2
        [102].15   // _
        [102].16   // _
        [102].17   // _
        [299]   // Indice dentro Origen Ruta 2
        [102].18   // _
        [300]   // Eqp Tolva Destino Ruta 1 y 2
        [102].19   // _
        [102].20   // _
        [301]   // Tiempo Total Ruta1
        [7].5   // Second Change
        [301].0   // CMD Intake
        [302]   // Tiempo Total Ruta2
        [102].21   // _
        [302].0   // State Intake
        [102].22   // _
        [302].1   // CLX Lin #2 o 3
        [102].23   // _
        [102].24   // _
        [102].25   // _
        [102].26   // _
        [102].27   // _
        [102].28   // _
        [102].29   // _
        [102].30   // _
        [102].31   // _
        [103].10   // _
        [103].11   // _
        [104].16   // _
        [104].17   // _
        [302].2   // CLX Lin #4
        [169]   // Password Interfaz 10 (HMI Serv.Aux)
        [321]   // Pop intake PanelView 1 - Item Guia
        [104].18   // _
        [131].1   // Batch Borrado
        [137]   // Rpt State
        [162]   // Usuario Interfaz 7 (HMI DMM)
        [303]   // Resp.(1=Term) (2=Reintentar)
        [163]   // Password Interfaz 7 (HMI DMM)
        [164]   // Usuario Interfaz 8 (HMI L1)
        [165]   // Password Interfaz 8 (HMI L1)
        [304]   // Resp.(1=Term) (2=Reintentar)
        [166]   // Usuario Interfaz 9 (HMI L2)
        [167]   // Password Interfaz 9 (HMI L2)
        [170]   // RSV Index Dos Arriba
        [305]   // Estado Ruta 1
        [305].0   // Toggle Batch Rx
        [175]   // Bind Result Rpt DMM
        [305].1   // Batch Erased
        [305].2   // Get Sprout Info
        [306]   // Estado Ruta 2
        [176]   // RSV Cmd Dosf Arriba
        [180]   // RSV Indx Desp
        [306].0   // Cmd InputMP
        [186]   // RSV Cmd Desp
        [190]   // Origen Index
        [191]   // Origen Old
        [193]   // Destino Futuro
        [204]   // Bind Result 21-30
        [205]   // Bind Result 31-40
        [206]   // Bind Result 41-50
        [8].0   // Alarma en Vacío Midis-Micros
        [8].17   // SQL Communication Error
        [8].18   // SQL Bad Answer Error
        [307]   // Flag
        [207]   // Bind Result 51-60
        [8].26   // SQL Folio Out Report Alarm
        [8].28   // MSG Timeout Alarm
        [208]   // Bind Result 61-70
        [2]   // System - Day
        [307].0   // Rev Input MP
        [8].29   // SQL Data Insert
        [9].0   // Cmd ON Master Inatke
        [9].1   // Cmd OFF Master Inatke
        [7].2   // Day Change
        [9].2   // Cmd ON Macros
        [8]   // Timestamp
        [9].3   // Cmd OFF Macros
        [209]   // Bind Result 71-80
        [9].4   // Cmd ON Mol y Mix
        [307].1   // Input MP OK
        [9].5   // Cmd OFF Mol y Mix
        [307].2   // Input Mp NOK
        [210]   // Import MP desde DB
        [11].20   // _
        [310]   // Numero de Guia
        [9].6   // Cmd ON Master Micros
        [9].7   // Cmd OFF Master Micros
        [11].21   // _
        [313]   // Pop Intake Def - Cod_MP
        [9].8   // Cmd ON Master Liq. Mixer
        [314]   // Check - Bin A
        [9].9   // Cmd OFF Master Liq. Mixer
        [9].10   // Cmd ON Quebrantado Linea 1
        [9].11   // Cmd OFF Quebrantado Linea 1
        [9].12   // Cmd ON Quebrantado Linea2
        [9].13   // Cmd OFF Quebrantado Linea 1
        [10]   // Fecha PLC Tx
        [211]   // Operador importó MP
        [10].2   // Master Despacho
        [212].0   // Enable LiveBin #1
        [315]   // Check - Bin B
        [11].22   // _
        [11].23   // _
        [11].24   // _
        [212].1   // Enable LiveBin #2
        [316]   // Check - Bin C
        [318]   // Interfaz
        [11].27   // _
        [13]   // PID Index
        [18].2   // RIO Abast
        [319]   // Sprout Counter old
        [18].5   // RIO Dosif
        [18].11   // RIO Desp
        [12]   // Total Eqp Fast
        [14].0   // Auto-Man PID Mol L1
        [14].1   // On-Off PID Mol L1
        [14].2   // Auto-Man PID Mol L2
        [14].3   // On-Off PID Mol L2
        [14].4   // Auto-Man PID Vent. Mol L1
        [14].5   // On-Off PID Vent. Mol L1
        [14].6   // Auto-Man PID Vent. Mol L2
        [20]   // Msg Code
        [14].7   // On-Off PID Vent. Mol L2
        [15].0   // Envío automático de Batch
        [212].2   // Enable LiveBin #3
        [15].2   // Botón envio batch L1
        [15].3   // Botón envio batch L2
        [15].4   // Linea 1 sin Macros
        [15].5   // Linea 2 sin Macros
        [15].6   // Pop-Up Desc. Previa Macros
        [15].7   // Ejecutar descarga previa
        [15].8   // Enable LB #1
        [15].9   // Enable LB #2
        [15].10   // Enable LB #3
        [15].11   // Faltan ing. Micros L1
        [15].15   // Start Molinos
        [213]   // Bind Result Bad
        [15].16   // Stop Molinos
        [22]   // Numero Bin
        [15].17   // Enable Molino #1
        [15].18   // Enable Molino #2
        [15].19   // Start Molino #1
        [214]   // User
        [23]   // Group
        [25]   // Old Answer
        [30]   // Msg Code
        [15].20   // Start Molino #2
        [30].0   // _
        [30].2   // _
        [15].21   // Auto-Man Molino #1
        [30].3   // _
        [15].22   // Auto-Man Molino #2
        [215]   // Cod_Error
        [220].2   // Start Molino
        [222]   // Linea
        [15].23   // Start LiveBins
        [15].24   // Stop LiveBins
        [15].25   // Start Transp. Lineas
        [15].26   // Stop Transp. Lineas
        [15].31   // Botón Sincronizar
        [223]   // Last_Folio
        [18].0   // Tension Ctrl Abast
        [30].4   // _
        [30].8   // _
        [18].1   // Modo Auto Abast
        [18].3   // Tension Ctrl Dosif
        [18].4   // Modo Auto Dosif
        [18].6   // Error Comm CNET PLT1
        [18].7   // Error Comm CNET PLT3
        [18].8   // Error Comm CNET Silos
        [18].9   // Modo Auto Desp
        [226]   // Cod_Error Recepccion
        [18].10   // Tension Ctrl Desp
        [18].14   // Alarma Voltaje TG-8
        [30].9   // _
        [18].15   // Alarma Asimetria TG-8
        [30].16   // _
        [18].16   // Cnet Dosif Falla
        [30].17   // _
        [30].18   // _
        [30].19   // _
        [18].17   // RIO Tolvas Falla
        [18].20   // PE Pelet. Sec. TCL_PS031
        [18].21   // PE Despacho TCL_PS032
        [18].24   // Cnet Pelet Falla
        [18].25   // Falla VDF Macros1
        [234]   // Interfaz Login
        [18].26   // Falla VDF Macros2
        [237]   // Fecha PLC Login
        [253]   // Password Interfaz 6 (HMI DMM)
        [324]   // Pop intake PanelView 1 - Bin A
        [325]   // Pop intake PanelView 1 - Bin B
        [326]   // Pop intake PanelView 1 - Bin C
        [328]   // Comando PV1
        [338]   // Comando PV2
        [254]   // Usuario Interfaz 7 (HMI DMM)
        [18].27   // Falla VDF Midis
        [18].28   // Falla VDF Micros
        [341]   // Additive 2 Setpoint
        [255]   // Password Interfaz 7 (HMI DMM)
        [256]   // Trigger Reporte DMM
        [21]   // Codigo Producto
        [342]   // Additive 1 Amount Counter
        [257]   // Bind Result Report DMM
        [258]   // TimeStamp Report DMM
        [0]   // System - Year
        [1]   // System - Month
        [3]   // System - Hour
        [4]   // System - Minute
        [5]   // System - Seconds
        [6]   // System - uSeconds
        [7].0   // Year Change
        [7].1   // Month Change
        [7].3   // Hour Change
        [24]   // Operador Answer
        [26]   // Folio Dosificandose Micros
        [7].4   // Minute Change
        [31].0   // _
        [259]   // TimeStamp Report DB
        [260].2   // Usuario no existe
        [260].3   // Bad Password
        [260].4   // Sin Permisos
        [343]   // Additive 2 Amount Counter
        [348]   // Comando PV3
        [280]   // PID Index from RSView
        [11]   // _
        [14]   // _
        [27]   // _
        [71]   // _
        [72]   // _
        [73]   // _
        [75]   // _
        [76]   // _
        [77]   // _
        [78]   // _
        [82]   // _
        [90]   // _
        [92]   // _
        [93]   // _
        [80]   // _
        [81]   // _
        [31].2   // _
        [31].3   // _
        [31].4   // _
        [31].8   // _
        [31].9   // _
        [31].16   // _
        [31].17   // _
        [31].18   // _
        [31].19   // _
        [32].8   // _
        [32].9   // _
        [32].10   // _
        [32].16   // _
        [32].17   // _
        [32].18   // _
        [32].19   // _
        [91].0   // _
        [91].1   // _
        [91].2   // _
        [91].3   // _
        [91].4   // _
        [91].5   // _
        [91].6   // _
        [94]   // _
        [95]   // _
        [96]   // _
        [97]   // _
        [98]   // _
        [100]   // _
        [100].0   // _
        [100].1   // _
        [100].2   // _
        [100].3   // _
        [100].4   // _
        [100].5   // _
        [100].6   // _
        [100].7   // _
        [100].8   // _
        [100].9   // _
        [101]   // _
        [101].0   // _
        [101].1   // _
        [101].2   // _
        [101].3   // _
        [101].4   // _
        [101].5   // _
        [101].6   // _
        [101].7   // _
        [101].8   // _
        [101].9   // _
        [102].0   // _
        [102].1   // _
        [102].2   // _
        [102].3   // _
        [102].4   // _
        [102].5   // _
        [102].6   // _
        [102].7   // _
        [102].8   // _
        [102].9   // _
        [103]   // _
        [103].0   // _
        [103].1   // _
        [103].2   // _
        [103].3   // _
        [103].4   // _
        [103].5   // _
        [103].6   // _
        [103].7   // _
        [103].8   // _
        [103].9   // _
        [104]   // _
        [104].0   // _
        [104].1   // _
        [104].3   // _
        [104].4   // _
        [104].5   // _
        [104].6   // _
        [104].7   // _
        [104].8   // _
        [104].9   // _
        [105]   // _
        [108].0   // _
        [108].1   // _
        [108].2   // _
        [108].3   // _
        [109]   // _
        [109].0   // _
        [109].1   // _
        [109].2   // _
        [109].3   // _
        [109].4   // _
        [109].5   // _
        [109].6   // _
        [171]   // _
        [172]   // _
        [173]   // _
        [174]   // _
        [177]   // _
        [178]   // _
        [179]   // _
        [181]   // _
        [182]   // _
        [183]   // _
        [184]   // _
        [185]   // _
        [187]   // _
        [188]   // _
        [189]   // _
        [192]   // _
        [398]   // OSR
        [10].1   // Master Dosificación
        [10].0   // Master Molienda
   vdf : VDFS[20] := ([1].ST := 66, [1].CMD := 8, [2].ST := 66, [3].ST := 66, [4].ST := 66, [5].ST := 66, [5].CMD := 8, [6].ST := 66, [6].FRQ_IN := 50.0, [6].FRQ_OUT := 50.0, [7].ST := 66, [8].ST := 66, [8].FRQ_IN := 21.0, [8].FRQ_OUT := 21.0, [9].ST := 66, [9].FRQ_IN := 10.0, [9].FRQ_OUT := 10.0, [10].ST := 66, [10].FRQ_IN := 20.0, [10].FRQ_OUT := 20.0, [11].ST := 66, [11].FRQ_IN := 30.0, [11].FRQ_OUT := 30.0, [11].Sincro_MSG := 1, [12].ST := 66, [12].FRQ_IN := 30.0, [12].FRQ_OUT := 30.0, [12].Sincro_MSG := 2, [13].ST := 66, [13].FRQ_IN := 30.0, [13].FRQ_OUT := 30.0, [13].Sincro_MSG := 2, [14].ST := 66, [14].FRQ_IN := 30.0, [14].FRQ_OUT := 30.0, [14].Sincro_MSG := 1);
   VDFidx : DINT;
END_VAR
